(* PLC project PLC_Programming_With_ST.project, TK TC6_v0200_Example3 v3.0 *)
(* stored: creationDateTime 2019-09-29T20:50:27.2524554, modificationDateTime 2020-05-23T11:25:38.4825215 *)

TYPE OnOff_ConstructorLIO : STRUCT
  Opened : BOOL;  (* Object is opened *)
  Closed : BOOL;  (* Object is closed *)
  PositionError : BOOL;  (* TRUE: Object has position error *)
END_STRUCT;
END_TYPE

TYPE dint8 : STRUCT
  first : DINT;
  second : DINT;
  third : DINT;
  fourth : DINT;
  fifth : DINT;
  sixth : DINT;
  seventh : DINT;
  eight : DINT;
END_STRUCT;
END_TYPE

TYPE MotorPump : STRUCT
  Running : BOOL;
  Fail : BOOL;
  DiffPress : BOOL;
END_STRUCT;
END_TYPE

TYPE MotorVentilator : STRUCT
  qMotor : BOOL;
  iOverheatProtection : BOOL;
  iOvercurrentProtection : BOOL;
  iMotorFailOther : BOOL;
  qLamp_Local : BOOL;
  iEmcy_Stop : BOOL := TRUE;
  iStart_Local : BOOL;
  iStop_Local : BOOL;
END_STRUCT;
END_TYPE

TYPE PrometnoSvjetlo : STRUCT
  ZelenoSvjetlo : BOOL;
  ZutoSvjetlo : BOOL;
  CrvenoSvjetlo : BOOL;
  PjesakovoDugme : BOOL;
END_STRUCT;
END_TYPE

{attribute 'qualified_only'}
VAR_GLOBAL  (* MixingTankGVL *)
  PushButtonStart : BOOL;  (* DIGITAL INPUT Naredba operator za start sustava *)
  PushButtonStop : BOOL;  (* DIGITAL INPUT Naredba operator za stop sustava *)
  Pump1StartCmd : BOOL;  (* DIGITAL OUTPUT Naredba automatike za start pumpe 1 *)
  Pump1StopCmd : BOOL;  (* DIGITAL OUTPUT Naredba automatike za stop pumpe 1 *)
  Pump1Running : BOOL;  (* DIGITAL INPUT Indikacija pokrenutog status pumpe 1 *)
  Pump2StartCmd : BOOL;  (* DIGITAL OUTPUT Naredba automatike za start pumpe 2 *)
  Pump2StopCmd : BOOL;  (* DIGITAL OUTPUT Naredba automatike za stop pumpe 2 *)
  Pump2Running : BOOL;  (* DIGITAL INPUT Indikacija pokrenutog status pumpe 2 *)
  DrainValveOpenCmd : BOOL;  (* DIGITAL OUTPUT Naredba automatike za otvaranje ventila za odvod *)
  DrainValveCloseCmd : BOOL;  (* DIGITAL OUTPUT Naredba automatike za zatvaranje ventila za odvod *)
  DrainValveClosed : BOOL;  (* DIGITAL INPUT Indikacija zatvorenog stanja odvodnog ventila *)
  DrainValveOpened : BOOL;  (* DIGITAL INPUT Indikacija otvorenog stanja odvodnog ventila *)
  TankLevel : REAL;  (* REAL VALUE Trenutna razina tanka u postocima *)
END_VAR

{attribute 'qualified_only'}
VAR_GLOBAL  (* Task02GVL *)
  HorizontalS1 : BOOL;  (* Configuration Inputs *)
  HorizontalS2 : BOOL;
  VerticalS1 : BOOL;
  VerticalS2 : BOOL;
  ManUp : BOOL;
  ManDown : BOOL;
  ManRight : BOOL;
  ManLeft : BOOL;
  ManUpRight : BOOL;
  ManUpLeft : BOOL;
  ManDownRight : BOOL;
  ManDownLeft : BOOL;
  Reset : BOOL;
  HorizontalRight : BOOL;  (* Outputs *)
  HorizontalLeft : BOOL;
  VerticalUp : BOOL;
  VerticalDown : BOOL;
END_VAR

{attribute 'qualified_only'}
VAR_GLOBAL  (* Task03GVL *)
  cfgPeriodTime : TIME := TIME#1m24s0ms;  (* Configuration *)
  cfgStartDirection : DINT := 0;
  TLight1Red : BOOL;  (* DIGITAL OUTPUT Activate red light traffic light 1 *)
  TLight1Yellow : BOOL;  (* DIGITAL OUTPUT Activate yellow light traffic light 1 *)
  TLight1Green : BOOL;  (* DIGITAL OUTPUT Activate green light traffic light 1 *)
  TLight2Red : BOOL;  (* DIGITAL OUTPUT Activate red light traffic light 2 *)
  TLight2Yellow : BOOL;  (* DIGITAL OUTPUT Activate yellow light traffic light 2 *)
  TLight2Green : BOOL;  (* DIGITAL OUTPUT Activate green light traffic light 2 *)
  TLight3Red : BOOL;  (* DIGITAL OUTPUT Activate red light traffic light 3 *)
  TLight3Yellow : BOOL;  (* DIGITAL OUTPUT Activate yellow light traffic light 3 *)
  TLight3Green : BOOL;  (* DIGITAL OUTPUT Activate green light traffic light 3 *)
  TLight4Red : BOOL;  (* DIGITAL OUTPUT Activate red light traffic light 4 *)
  TLight4Yellow : BOOL;  (* DIGITAL OUTPUT Activate yellow light traffic light 4 *)
  TLight4Green : BOOL;  (* DIGITAL OUTPUT Activate green light traffic light 4 *)
END_VAR



{attribute 'qualified_only'}
VAR_GLOBAL  (* Task06GVL *)
  JoyUp : BOOL;  (* Configuration Inputs *)
  JoyDown : BOOL;
  JoyRight : BOOL;
  JoyLeft : BOOL;
  JoyUpRight : BOOL;
  JoyUpLeft : BOOL;
  JoyDownRight : BOOL;
  JoyDownLeft : BOOL;
  EmcyStop : BOOL;
  RightLimit : BOOL;
  LeftLimit : BOOL;
  UpperLimit : BOOL;
  LowerLimit : BOOL;
  MotorLeft : BOOL;  (* Outputs *)
  MotorRight : BOOL;
  CraneDown : BOOL;
  CraneUp : BOOL;
END_VAR





PROGRAM FOR_Loop
  VAR CONSTANT
    ARR_SIZE : USINT := 9;  (* Size of the cube *)
  END_VAR
  VAR
    vType : USINT := 0;
    data : ARRAY[0..ARR_SIZE, 0..ARR_SIZE] OF BOOL;  (* Data for iteration *)
    i : USINT;  (* Iterators *)
    j : USINT;  (* Iterators *)
    vIncStep : BOOL;  (* Support functionalities *)
    vDecStep : BOOL;
    vStepTime : TIME := TIME#1s0ms;
    vStepTimeChange : TIME := TIME#100ms;
    Stepper : BLINK;
  END_VAR

            CASE vType OF
	0: (*FOR LOOP*)
		(*Loop over everything, set always to inverse*)
		FOR i:=0 TO ARR_SIZE DO
			(*Go through all the columns of this row*)
			FOR j:=0 TO ARR_SIZE DO
				data[i,j] := NOT data[i,j];
			END_FOR
		END_FOR
		
	1: (*WHILE LOOP*)
		(*Loop over everything, set always to inverse*)
		WHILE i <= ARR_SIZE DO
			(*Go trough all the columns*)
			WHILE j <= ARR_SIZE DO
				data[i,j] := NOT data[i,j];
				j := j + 1;
			END_WHILE
			j := 0;
			(*After each column, increase row by 1*)
			i := i + 1;			
		END_WHILE
		(*If we ended up here, that means we went throguh all the elements,
		so we can reset and start all over*)
		i := 0;
		j := 0;
	
	2: (*Repeat loop*)
		(*Repeat loop executes atleast once*)
		REPEAT

			REPEAT
				data[i,j] := NOT data[i,j];
				j := j + 1;
			UNTIL
				j > ARR_SIZE
			END_REPEAT
			j := 0;
			i := i + 1;
		UNTIL
			i > ARR_SIZE
		END_REPEAT
		i := 0;
		j := 0;
		
	3: (*Cycle loop on 100 ms*)
		data[i,j] := NOT data[i,j];
		j := j + 1;
		IF j > ARR_SIZE THEN
			j:=0;
			i := i + 1;
			IF i > ARR_SIZE THEN
				i := 0;
			END_IF
		END_IF
		
	4: (*Pulse/Trigger loop*)
		IF Stepper.OUT THEN
			data[i,j] := NOT data[i,j];
			j := j + 1;
			IF j > ARR_SIZE THEN
				j:=0;
				i := i + 1;
				IF i > ARR_SIZE THEN
					i := 0;
				END_IF
			END_IF
		END_IF
	
	5: (*Reset - Set all to false*)
		MEMUtils.MemSet(ADR(data),0, SIZEOF(data));
END_CASE

(*Support functionality*)
(*Step speed*)
IF vIncStep THEN
	vStepTime := LIMIT(T#0.1S, vStepTime + vStepTimeChange, T#10S);
ELSIF vDecStep THEN
	vStepTime := LIMIT(T#0.1S, vStepTime - vStepTimeChange, T#10S);
END_IF
Stepper(ENABLE:= TRUE, TIMELOW:= vStepTime, TIMEHIGH:= T#100MS);
          
END_PROGRAM

FUNCTION_BLOCK CollisionDetection
  VAR_INPUT
    xcor1 : REAL := 0;  (* X Coordinate of object 1 *)
    ycor1 : REAL := 0;  (* Y Coordinate of object 1 *)
    height1 : REAL := 0;  (* Height of object 1 *)
    width1 : REAL := 0;  (* Width of object 1 *)
    xcor2 : REAL := 0;  (* X Coordinate of object 2 *)
    ycor2 : REAL := 0;  (* Y Coordinate of object 2 *)
    height2 : REAL := 0;  (* Height of object 1 *)
    width2 : REAL := 0;  (* Width of object 1 *)
  END_VAR
  VAR_OUTPUT
    isCollision : BOOL := FALSE;
  END_VAR

            IF xcor1 < (xcor2 + width2) AND
   (xcor1 + width1) > xcor2 AND
   ycor1 < (ycor2 + height2) AND
  ( height1 + ycor1) > ycor2 THEN
   isCollision := TRUE;
ELSE
	isCollision := FALSE;
END_IF
          
END_FUNCTION_BLOCK

FUNCTION CONCAT2 : STRING
  VAR_INPUT
    STR : ARRAY[0..19] OF STRING;  (* String array filled with characters to concatenate *)
  END_VAR
  VAR
    vStr : STRING := '';
    i : UINT := 0;
    vSize : UINT;
  END_VAR

            vStr := '';
vSize :=(SIZEOF(STR)/81);

FOR i:=0 TO vSize - 1 BY 1 DO
	IF STR[i] <> '' THEN
		vStr := CONCAT(vStr, STR[i]);
	END_IF
END_FOR
CONCAT2 := vStr;
          
END_FUNCTION

PROGRAM PLC_PRG_1
  VAR
    Start_Switch : BOOL;
    Bottle : BOOL;
    UpperLimitSwitch : BOOL := TRUE;
    ConveyorBeltPut : BOOL;
    ConveyorBeltSimPut : TON;
    TimeSimConvey : TIME := TIME#2s0ms;
    MotorDown : BOOL;
    LowerLimitSwitch : BOOL;
    MotorUp : BOOL;
    MovingDownSim : TON;
    TimeDownSim : TIME := TIME#4s0ms;
    ElapsedTimeDown : TIME;
    TimeCheck : TIME := TIME#0ms;
    BottleStamped : BOOL;
    MovingUpSim : TON;
    TimeUpSim : TIME := TIME#4s0ms;
    ElapsedTimeUp : TIME;
    ConveyorBeltRemove : BOOL;
    ConveyorBeltRemoveSim : TON;
    ConveyorBeltMotor : BOOL;
  END_VAR

            IF Start_Switch THEN

	(* Putting new bottle under the marker if there isnt any *)
	IF NOT Bottle AND UpperLimitSwitch THEN
		ConveyorBeltPut := TRUE;
	ELSE
		ConveyorBeltPut := FALSE;
	END_IF;

	(*Simulating the conveyor belt putting new bottle in*)
	ConveyorBeltSimPut(IN:= ConveyorBeltPut, PT:= TimeSimConvey);

	IF ConveyorBeltSimPut.Q THEN
		Bottle := TRUE;
	END_IF;

	MotorDown := Bottle AND NOT LowerLimitSwitch AND NOT MotorUp;
	(*Simulating the movement of the motor down and engaging the limit switches*)
	MovingDownSim(IN := MotorDown, PT := TimeDownSim, ET => ElapsedTimeDown);

	IF MovingDownSim.ET <> TimeCheck THEN
		UpperLimitSwitch := FALSE;
	END_IF;

	IF MovingDownSim.Q THEN
		LowerLimitSwitch := TRUE;
		BottleStamped :=TRUE;
	END_IF;

	MotorUp := BottleStamped AND NOT UpperLimitSwitch AND NOT MotorDown;
	(*Simulating the movement of the motor up and engaging the limit switches*)
	MovingUpSim(IN := MotorUp,PT := TimeUpSim, ET=>ElapsedTimeUp);

	IF MovingUpSim.ET <> TimeCheck THEN
		LowerLimitSwitch := FALSE;
	END_IF;

	IF MovingUpSim.Q THEN
		UpperLimitSwitch := TRUE;
	END_IF;

	IF BottleStamped AND UpperLimitSwitch THEN
		ConveyorBeltRemove := TRUE;
		(*Simulating the rotation of the conveyor and removing the bottles that is stamped*)
		ConveyorBeltRemoveSim(IN := ConveyorBeltRemove, PT := TimeSimConvey );
		IF ConveyorBeltRemoveSim.Q THEN
			Bottle := FALSE;
			BottleStamped := FALSE;
		END_IF;
	ELSE
		ConveyorBeltRemove := FALSE;
	END_IF;

	ConveyorBeltMotor := ConveyorBeltRemove OR ConveyorBeltPut;

END_IF;
(*
IF Start_Switch THEN

	IF  UpperLimitSwitch
		AND NOT LowerLimitSwitch
		AND NOT CylinderUpMotor
		THEN
			CylinderDownMotor := TRUE;
	END_IF;

	UpperLSWDelay(IN:=CylinderDownMotor, PT:=T#10S);
	IF 	UpperLSWDelay.Q
	THEN
		LowerLimitSwitch := TRUE;
	END_IF;

	IF  LowerLimitSwitch
	THEN
		CylinderDownMotor:= FALSE;
	END_IF;

	IF 	UpperLimitSwitch
	THEN
		CylinderUpMotor := FALSE;
	END_IF;

	IF 			 LowerLimitSwitch
		AND NOT  UpperLimitSwitch
	THEN
				 CylinderUpMotor := TRUE;
	END_IF;
	
	LowerLSWDelay(IN:=CylinderUpMotor, PT:=T#10S);
	IF 	LowerLSWDelay.Q
	THEN
		UpperLimitSwitch := TRUE;
	END_IF;

	IF UpperLimitSwitch
	THEN
		LowerLimitSwitch := FALSE;
	ELSE IF LowerLimitSwitch
	THEN
 	UpperLimitSwitch:FALSE;
	END_IF;

END_IF;
*)

          
END_PROGRAM

FUNCTION_BLOCK Motor_Model
  VAR_INPUT
    CBActivated : BOOL := FALSE;
    LineVoltage : REAL := 440;
    cfgNominalPower : REAL := 12;  (* kW *)
    cfgPowerFactor : REAL := 0.83;
    Frequency : REAL := 60;
    cfgNoOfPoles : DINT := 4;
    cfgSpeedUpRate : REAL := 800;
    cfgSpeedDownRate : REAL := 800;
    simShortCircuit : BOOL := FALSE;
  END_VAR
  VAR_OUTPUT
    CurrentL1 : LREAL := 0;
    CurrentL2 : LREAL := 0;
    CurrentL3 : LREAL := 0;
    Speed : REAL := 0;
    Status : ARRAY[0..10] OF BOOL;
  END_VAR
  VAR
    vNs : REAL;
    vPhaseCurrent : REAL := 0;
    SpeedRamp : RAMP_REAL;
    SpeedBlink : BLINK;
    vBlinkTime : REAL;
    vBlinker : BOOL;
    vApparentPower_kVA : REAL;
  END_VAR

            Status[0] := CBActivated;;

vApparentPower_kVA := cfgNominalPower/(3*cfgPowerFactor);

vPhaseCurrent := (vApparentPower_kVA*1000)/LineVoltage;

CurrentL1 := (vPhaseCurrent/SQRT(3)+(BOOL_TO_REAL(simShortCircuit)*250))*BOOL_TO_REAL(Status[0]);
CurrentL2 := (vPhaseCurrent/SQRT(3)+(BOOL_TO_REAL(simShortCircuit)*250))*BOOL_TO_REAL(Status[0]);
CurrentL3 := (vPhaseCurrent/SQRT(3)+(BOOL_TO_REAL(simShortCircuit)*250))*BOOL_TO_REAL(Status[0]);

vNs := ((120 *Frequency)/DINT_TO_REAL(cfgNoOfPoles))*BOOL_TO_REAL(Status[0]);

SpeedRamp(
	IN:= vNs, 
	ASCEND:= cfgSpeedUpRate, 
	DESCEND:= cfgSpeedDownRate, 
	TIMEBASE:= T#2S, 
	OUT=>Speed);
	
vBlinkTime := 100000/MAX(1,Speed);

SpeedBlink(ENABLE:= vBlinkTime < 100000, TIMELOW:= REAL_TO_TIME(vBlinkTime), TIMEHIGH:= REAL_TO_TIME(vBlinkTime), OUT=> Status[1]);
          
END_FUNCTION_BLOCK

FUNCTION_BLOCK On_Off_Constructor
  VAR_INPUT
    iOpenedFB : BOOL;  (* IO Open signal feedback from the valve *)
    iClosedFB : BOOL;  (* IO Close signal feedback from the valve *)
    cfgPositionErrorDelay : TIME := TIME#10s0ms;  (* Position error alarm delay *)
    cfgFBs : DWORD := 3;  (* B0 - Opened signal in use, B1 - Closed signal in use *)
  END_VAR
  VAR_OUTPUT
    LIO : OnOff_ConstructorLIO;  (* Communication structure to higher logic *)
    HMI : OnOff_ConstructorLIO;  (* Communication structure to HMI *)
  END_VAR
  VAR
    PositionErrorDelay : TON;  (* Position error alarm delay *)
    vPositionErrorOld : BOOL;  (* Event memory: Position error *)
    vOpenedOld : BOOL;  (* Event memory: Opened *)
    vClosedOld : BOOL;  (* Event memory: Closed *)
  END_VAR

            (* Handle IOs depending on CFG *)
IF cfgFBs.0 AND cfgFBs.1 THEN
	LIO.Closed := iClosedFB;
	LIO.Opened := iOpenedFB;
ELSIF cfgFBs.0 THEN
	LIO.Closed := NOT iOpenedFB;
	LIO.Opened := iOpenedFB;
ELSIF cfgFBs.1 THEN
	LIO.Closed := iClosedFB;
	LIO.Opened := NOT iClosedFB;
ELSE
	(* Invalid configuration *)
END_IF;

(* Alarm management *)
(* Position error *)
PositionErrorDelay(
	IN:= LIO.Closed AND LIO.Opened OR NOT (LIO.Closed OR LIO.Opened),
	PT:= cfgPositionErrorDelay,
	Q  => LIO.PositionError);

(* Event management *)
(* Breaker opened *)
IF LIO.Opened AND NOT vOpenedOld THEN
	(* Call event *)
END_IF

(* Breaker closed *)
IF LIO.Closed AND NOT vClosedOld THEN
	(* Call event *)
END_IF
(* Position error *)
IF LIO.PositionError AND NOT vPositionErrorOld THEN
	(* Call event *)
END_IF

(* Communicate status to HMI *)	
HMI := LIO;


 
          
END_FUNCTION_BLOCK

FUNCTION_BLOCK OnOffValve_Model
  VAR_INPUT
    OpenCmd : BOOL;  (* Command to open the valve *)
    CloseCmd : BOOL;  (* Command to close the valve *)
    cfgOpeningTime : TIME := TIME#5s0ms;  (* Time it take to open the valve *)
    cfgClosingTime : TIME := TIME#5s0ms;  (* Time it take to close the valve *)
    simOpenFail : BOOL;  (* Simulated open fail when true *)
    simCloseFail : BOOL;  (* Simulated close fail when true *)
  END_VAR
  VAR_OUTPUT
    Opened : BOOL;
    Closed : BOOL;
  END_VAR
  VAR
    OpenTime : TON;
    CloseTime : TON;
  END_VAR

            (* Description of action:
If the open/close signal comes the valve opens/closes in designated time *)

OpenTime(IN:= OpenCmd AND NOT Opened, PT:=cfgOpeningTime);
CloseTime(IN:= CloseCmd AND NOT Closed, PT:=cfgClosingTime);

IF Opened AND CloseCmd THEN
	Opened := FALSE;
ELSIF OpenTime.Q AND NOT simOpenFail THEN
	Opened := TRUE;
END_IF

IF Closed AND OpenCmd THEN
	Closed := FALSE;
ELSIF CloseTime.Q AND NOT simCloseFail THEN
	Closed := TRUE;
END_IF
          
END_FUNCTION_BLOCK

FUNCTION_BLOCK OnOffValve_Object
  VAR_INPUT
    iOpenedFB : BOOL;  (* IO Open signal feedback from the valve *)
    iClosedFB : BOOL;  (* IO Close signal feedback from the valve *)
    OpenAutoCmd : BOOL;  (* Open cmd from program logic *)
    CloseAutoCmd : BOOL;  (* Close cmd from program logic *)
    OpenCmdHMI : BOOL;  (* Open cmd from HMI *)
    CloseCmdHMI : BOOL;  (* Close cmd from HMI *)
    SetToAuto : BOOL;  (* Sets valve control to auto mode *)
    SetToMan : BOOL;  (* Sets valve control to manual mode *)
    cfgOpenFailDelay : TIME := TIME#6s0ms;  (* Open fail delay *)
    cfgCloseFailDelay : TIME := TIME#6s0ms;  (* Close fail delay *)
    cfgPositionErrorDelay : TIME := TIME#10s0ms;  (* Position error delay *)
    cfgFBs : DWORD := 16#3;  (* B0 - Opened signal in use, B1 - Closed signal in use *)
  END_VAR
  VAR_OUTPUT
    ValveStatus : ARRAY[1..20] OF DINT;  (* 1:Open/Closed/InTransit, 2:OpenFail, 3:CloseFail, 4:FBError, 5:Control Position, 6:OpenCmd, 7:CloseCmd *)
    ValveIcon : STRING;
    qOpenCmd : BOOL;  (* IO Open command signal *)
    qCloseCmd : BOOL;  (* IO Close command signal *)
  END_VAR
  VAR
    ObjConstructor : On_Off_Constructor;  (* Base building block of this object *)
    OpenFail : TON;
    CloseFail : TON;
    vControlPosition : DINT;
    vOpenCmd : BOOL;
    vCloseCmd : BOOL;
  END_VAR

            (* Handle base constructor *)
ObjConstructor(
	iOpenedFB := iOpenedFB,
	iClosedFB := iClosedFB,
	cfgPositionErrorDelay := cfgPositionErrorDelay,
	cfgFBs := cfgFBs);

(* Control position *)
(* Auto/Man setting should be rtrig or non holding button *)
IF SetToAuto AND NOT SetToMan THEN
	vControlPosition := 1;
ELSIF SetToMan THEN
	vControlPosition := 0;
END_IF

IF NOT(OpenFail.Q OR CloseFail.Q) THEN
	IF vControlPosition = 1 THEN
		vOpenCmd := (vOpenCmd OR OpenAutoCmd) AND NOT ObjConstructor.LIO.Opened;
		vCloseCmd := (vCloseCmd OR CloseAutoCmd) AND NOT ObjConstructor.LIO.Closed;
	ELSIF vControlPosition = 0 THEN
		vOpenCmd := (vOpenCmd OR OpenCmdHMI) AND NOT ObjConstructor.LIO.Opened;
		vCloseCmd := (vCloseCmd OR CloseCmdHMI) AND NOT ObjConstructor.LIO.Closed;
	ELSE
		vOpenCmd := FALSE;
		vCloseCmd := FALSE;	
	END_IF
ELSE
		vOpenCmd := FALSE;
		vCloseCmd := FALSE;		
END_IF

OpenFail(IN:= vOpenCmd AND NOT ObjConstructor.LIO.Opened, PT:= cfgOpenFailDelay);
CloseFail(IN:= vCloseCmd AND NOT ObjConstructor.LIO.Closed, PT:= cfgCloseFailDelay);

qOpenCmd := vOpenCmd AND NOT (OpenFail.Q OR ObjConstructor.LIO.Opened OR ObjConstructor.LIO.PositionError);
qCloseCmd := vCloseCmd AND NOT (CloseFail.Q OR ObjConstructor.LIO.Closed OR ObjConstructor.LIO.PositionError);

ValveStatus[1] := BOOL_TO_DINT(ObjConstructor.LIO.Opened) + 2*BOOL_TO_DINT(ObjConstructor.LIO.Closed);
ValveStatus[2] := BOOL_TO_DINT(OpenFail.Q);
ValveStatus[3] := BOOL_TO_DINT(CloseFail.Q);
ValveStatus[4] := BOOL_TO_DINT(ObjConstructor.LIO.PositionError);
ValveStatus[5] := vControlPosition;
ValveStatus[6] := BOOL_TO_DINT(qOpenCmd);
ValveStatus[7] := BOOL_TO_DINT(qCloseCmd);

IF ValveStatus[1] = 1 THEN
	ValveIcon := 'Valve1';
ELSIF ValveStatus[1] = 2 THEN
	ValveIcon := 'Valve2';
ELSE
	ValveIcon := 'Valve3';
END_IF


          
END_FUNCTION_BLOCK

PROGRAM PriorityPOU
  VAR
    SortPriority : PrioritySort;
    SwapSequence1 : Swapper;
    SwapSequence2 : Swapper;
    FPSequenceChangeTimer : TON;
    vEngineSequence : dint8;
    vFPSequence : dint8;
    vPPSequence : dint8;
    vModeManagerSequence : dint8;
    vApplyNewSequence : BOOL;
    vApplyButtonPermission : BOOL;
    vNewSequence : dint8;
    vSequenceIsSame : BOOL;
    vValidStartSequenceSum : LREAL;
    vEngineSequenceSum : LREAL;
    vFPSequenceSum : LREAL;
    vFPSequenceInvalid : BOOL;
    vApplyButton2Permission : BOOL;
  END_VAR
  VAR RETAIN
    vRestarted : BOOL := FALSE;
    vInvalidSequence : BOOL;
  END_VAR

            
IF NOT vRestarted OR vInvalidSequence THEN
	(* Reinitialize priority list *)
	vEngineSequence.first := 1;
	vEngineSequence.second := 2;
	vEngineSequence.third  := 3;
	vEngineSequence.fourth := 4;
	vEngineSequence.fifth := 5;
	vEngineSequence.sixth := 6;
	vEngineSequence.seventh := 7;
	vEngineSequence.eight := 8;
	vFPSequence := vEngineSequence;
	vRestarted := TRUE;
END_IF

(* Determine correct sequence sum *)
vValidStartSequenceSum := EXPT(2,1)
						+ EXPT(2,2)
						+ EXPT(2,3)
                        + EXPT(2,4)
						+ EXPT(2,5)
						+ EXPT(2,6)
						+ EXPT(2,7)
						+ EXPT(2,8);

(* Constantly check engine sequence to make sure it is correct *)
vEngineSequenceSum := EXPT(2,vEngineSequence.first)
					+ EXPT(2,vEngineSequence.second)
					+ EXPT(2,vEngineSequence.third)
                    + EXPT(2,vEngineSequence.fourth)
				    + EXPT(2,vEngineSequence.fifth)
				    + EXPT(2,vEngineSequence.sixth)
					+ EXPT(2,vEngineSequence.seventh)
					+ EXPT(2,vEngineSequence.eight);
					
vInvalidSequence := vEngineSequenceSum <> vValidStartSequenceSum;

(* Faceplate start sequence handling *)
vSequenceIsSame :=  vEngineSequence.first = vFPSequence.first
				AND vEngineSequence.second = vFPSequence.second
				AND vEngineSequence.third = vFPSequence.third
				AND vEngineSequence.fourth = vFPSequence.fourth
				AND vEngineSequence.fifth = vFPSequence.fifth
				AND vEngineSequence.sixth = vFPSequence.sixth
				AND vEngineSequence.seventh = vFPSequence.seventh
				AND vEngineSequence.eight = vFPSequence.eight;

vFPSequenceSum := EXPT(2,vFPSequence.first)
				+ EXPT(2,vFPSequence.second)
				+ EXPT(2,vFPSequence.third)
                + EXPT(2,vFPSequence.fourth)
				+ EXPT(2,vFPSequence.fifth)
				+ EXPT(2,vFPSequence.sixth)
				+ EXPT(2,vFPSequence.seventh)
				+ EXPT(2,vFPSequence.eight);
				
vFPSequenceInvalid := vFPSequenceSum <> vValidStartSequenceSum;	
			
FPSequenceChangeTimer(IN:= NOT vSequenceIsSame OR vFPSequenceInvalid, PT:=T#15S);
IF FPSequenceChangeTimer.Q THEN
	vFPSequence := vEngineSequence;
END_IF;	
		
(* Swapper function 
- swaps places with the selected number*)
SwapSequence1(Enable:= NOT vSequenceIsSame, SequenceIN:= vFPSequence, SequenceOut => vFPSequence);

(* Functionality:
- Takes care of reseting invalid seq
- Applies requests
- converts to engine format
*)
SortPriority(
	EngineSequenceIN := vEngineSequence,
	RequestSequence1:= vFPSequence,
	RequestSequence1Permission:= NOT vFPSequenceInvalid,
	RequestSequence1Apply:= vApplyNewSequence,
	RequestSequence2:= vPPSequence,
	RequestSequence2Permission:= FALSE,
	RequestSequence2Apply:= FALSE,
	RequestSequence1ApplyPermission=> vApplyButtonPermission,
	RequestSequence2ApplyPermission=> vApplyButton2Permission,
	RequestSequence1OUT=> vFPSequence,
	RequestSequence2OUT=> vPPSequence,
	EngineSequenceOUT=> vEngineSequence);

          
END_PROGRAM

FUNCTION_BLOCK PrioritySort
  VAR_INPUT
    EngineSequenceIN : dint8;
    RequestSequence1 : dint8;
    RequestSequence1Permission : BOOL;
    RequestSequence1Apply : BOOL;
    RequestSequence2 : dint8;
    RequestSequence2Permission : BOOL;
    RequestSequence2Apply : BOOL;
  END_VAR
  VAR_OUTPUT
    RequestSequence1ApplyPermission : BOOL;
    RequestSequence2ApplyPermission : BOOL;
    RequestSequence1OUT : dint8;
    RequestSequence2OUT : dint8;
    EngineSequenceOUT : dint8;
  END_VAR
  VAR
    v1stSeqDifferent : BOOL;
    v2ndSeqDifferent : BOOL;
  END_VAR

            (* Compare sequences *)
v1stSeqDifferent := RequestSequence1.first <> EngineSequenceIN.first
				OR  RequestSequence1.second <> EngineSequenceIN.second
				OR  RequestSequence1.third <> EngineSequenceIN.third
				OR  RequestSequence1.fourth <> EngineSequenceIN.fourth
				OR  RequestSequence1.fifth <> EngineSequenceIN.fifth
				OR  RequestSequence1.sixth <> EngineSequenceIN.sixth
				OR  RequestSequence1.seventh <> EngineSequenceIN.seventh
				OR  RequestSequence1.eight <> EngineSequenceIN.eight;

v2ndSeqDifferent := RequestSequence2.first <> EngineSequenceIN.first
				OR  RequestSequence2.second <> EngineSequenceIN.second
				OR  RequestSequence2.third <> EngineSequenceIN.third
				OR  RequestSequence2.fourth <> EngineSequenceIN.fourth
				OR  RequestSequence2.fifth <> EngineSequenceIN.fifth
				OR  RequestSequence2.sixth <> EngineSequenceIN.sixth
				OR  RequestSequence2.seventh <> EngineSequenceIN.seventh
				OR  RequestSequence2.eight <> EngineSequenceIN.eight;

IF v1stSeqDifferent AND RequestSequence1Permission AND RequestSequence1Apply THEN
	EngineSequenceOUT := RequestSequence1;
	RequestSequence2OUT := RequestSequence1;
	
ELSIF v2ndSeqDifferent AND RequestSequence2Permission AND RequestSequence2Apply THEN
	EngineSequenceOUT := RequestSequence2;
	RequestSequence1OUT := RequestSequence2;
	
ELSE
	(* Basically do nothing, copy parameters *)
	EngineSequenceOUT := EngineSequenceIN;
	RequestSequence1OUT := RequestSequence1;
	RequestSequence2OUT := RequestSequence2;
END_IF

(* Send out permissions *)
RequestSequence1ApplyPermission:= RequestSequence1Permission AND NOT RequestSequence2Apply;
RequestSequence2ApplyPermission:= RequestSequence2Permission AND NOT RequestSequence1Apply;
          
END_FUNCTION_BLOCK

FUNCTION_BLOCK Swapper
  VAR_INPUT
    Enable : BOOL;
    SequenceIn : dint8;
  END_VAR
  VAR_OUTPUT
    SequenceOut : dint8;
  END_VAR
  VAR
    vTemp : DINT;
  END_VAR

            IF Enable THEN
	(* Check if any of the positions have changed values *)
	IF SequenceIN.first <> SequenceOut.first THEN
		(* If this position changed, save the old position and apply new one to its place *)
		vTemp:= SequenceOut.first;
		SequenceOut.first := SequenceIN.first;
		(* Find the position where the same number is and write temp there
		but skip this position *)
		IF SequenceIN.first = SequenceOut.second THEN
			SequenceOut.second := vTemp;
		ELSIF SequenceIN.first = SequenceOut.third THEN
			SequenceOut.third := vTemp;
		ELSIF SequenceIN.first = SequenceOut.fourth THEN
			SequenceOut.fourth := vTemp;
		ELSIF SequenceIN.first = SequenceOut.fifth THEN
			SequenceOut.fifth := vTemp;
		ELSIF SequenceIN.first = SequenceOut.sixth THEN
			SequenceOut.sixth := vTemp;
		ELSIF SequenceIN.first = SequenceOut.seventh THEN
			SequenceOut.seventh := vTemp;
		ELSIF SequenceIN.first = SequenceOut.eight THEN
			SequenceOut.eight := vTemp;
		END_IF
	ELSIF SequenceIN.second <> SequenceOut.second THEN
		vTemp:= SequenceOut.second;
		SequenceOut.second := SequenceIN.second;
		(* Find the index where the same number is and write temp there
		but skip this position *)
		IF SequenceIN.second = SequenceOut.first THEN
			SequenceOut.first := vTemp;
		ELSIF SequenceIN.second = SequenceOut.third THEN
			SequenceOut.third := vTemp;
		ELSIF SequenceIN.second = SequenceOut.fourth THEN
			SequenceOut.fourth := vTemp;
		ELSIF SequenceIN.second = SequenceOut.fifth THEN
			SequenceOut.fifth := vTemp;
		ELSIF SequenceIN.second = SequenceOut.sixth THEN
			SequenceOut.sixth := vTemp;
		ELSIF SequenceIN.second = SequenceOut.seventh THEN
			SequenceOut.seventh := vTemp;
		ELSIF SequenceIN.second = SequenceOut.eight THEN
			SequenceOut.eight := vTemp;
		END_IF
	ELSIF SequenceIN.third <> SequenceOut.third THEN
			vTemp:= SequenceOut.third;
		SequenceOut.third := SequenceIN.third;
		(* Find the index where the same number is and write temp there
		but skip this position *)
		IF SequenceIN.third = SequenceOut.first THEN
			SequenceOut.first := vTemp;
		ELSIF SequenceIN.third = SequenceOut.second THEN
			SequenceOut.second := vTemp;
		ELSIF SequenceIN.third = SequenceOut.fourth THEN
			SequenceOut.fourth := vTemp;
		ELSIF SequenceIN.third = SequenceOut.fifth THEN
			SequenceOut.fifth := vTemp;
		ELSIF SequenceIN.third = SequenceOut.sixth THEN
			SequenceOut.sixth := vTemp;
		ELSIF SequenceIN.third = SequenceOut.seventh THEN
			SequenceOut.seventh := vTemp;
		ELSIF SequenceIN.third = SequenceOut.eight THEN
			SequenceOut.eight := vTemp;
		END_IF
	ELSIF SequenceIN.fourth <> SequenceOut.fourth THEN
			vTemp:= SequenceOut.fourth;
		SequenceOut.fourth := SequenceIN.fourth;
		(* Find the index where the same number is and write temp there
		but skip this position *)
		IF SequenceIN.third = SequenceOut.first THEN
			SequenceOut.first := vTemp;
		ELSIF SequenceIN.fourth = SequenceOut.second THEN
			SequenceOut.second := vTemp;
		ELSIF SequenceIN.fourth = SequenceOut.third THEN
			SequenceOut.third := vTemp;
		ELSIF SequenceIN.fourth = SequenceOut.fifth THEN
			SequenceOut.fifth := vTemp;
		ELSIF SequenceIN.fourth = SequenceOut.sixth THEN
			SequenceOut.sixth := vTemp;
		ELSIF SequenceIN.fourth = SequenceOut.seventh THEN
			SequenceOut.seventh := vTemp;
		ELSIF SequenceIN.fourth = SequenceOut.eight THEN
			SequenceOut.eight := vTemp;
		END_IF
	ELSIF SequenceIN.fifth <> SequenceOut.fifth THEN
			vTemp:= SequenceOut.fifth;
		SequenceOut.fifth := SequenceIN.fifth;
		(* Find the index where the same number is and write temp there
		but skip this position *)
		IF SequenceIN.fifth = SequenceOut.first THEN
			SequenceOut.first := vTemp;
		ELSIF SequenceIN.fifth = SequenceOut.second THEN
			SequenceOut.second := vTemp;
		ELSIF SequenceIN.fifth = SequenceOut.third THEN
			SequenceOut.third := vTemp;
		ELSIF SequenceIN.fifth = SequenceOut.fourth THEN
			SequenceOut.fourth := vTemp;
		ELSIF SequenceIN.fifth = SequenceOut.sixth THEN
			SequenceOut.sixth := vTemp;
		ELSIF SequenceIN.fifth = SequenceOut.seventh THEN
			SequenceOut.seventh := vTemp;
		ELSIF SequenceIN.fifth = SequenceOut.eight THEN
			SequenceOut.eight := vTemp;
		END_IF
	ELSIF SequenceIN.sixth <> SequenceOut.sixth THEN
			vTemp:= SequenceOut.sixth;
		SequenceOut.sixth := SequenceIN.sixth;
		(* Find the index where the same number is and write temp there
		but skip this position *)
		IF SequenceIN.sixth = SequenceOut.first THEN
			SequenceOut.first := vTemp;
		ELSIF SequenceIN.sixth = SequenceOut.second THEN
			SequenceOut.second := vTemp;
		ELSIF SequenceIN.sixth = SequenceOut.third THEN
			SequenceOut.third := vTemp;
		ELSIF SequenceIN.sixth = SequenceOut.fourth THEN
			SequenceOut.fourth := vTemp;
		ELSIF SequenceIN.sixth = SequenceOut.fifth THEN
			SequenceOut.fifth := vTemp;
		ELSIF SequenceIN.sixth = SequenceOut.seventh THEN
			SequenceOut.seventh := vTemp;
		ELSIF SequenceIN.sixth = SequenceOut.eight THEN
			SequenceOut.eight := vTemp;
		END_IF
	ELSIF SequenceIN.seventh <> SequenceOut.seventh THEN
			vTemp:= SequenceOut.seventh;
		SequenceOut.seventh := SequenceIN.seventh;
		(* Find the index where the same number is and write temp there
		but skip this position *)
		IF SequenceIN.seventh = SequenceOut.first THEN
			SequenceOut.first := vTemp;
		ELSIF SequenceIN.seventh = SequenceOut.second THEN
			SequenceOut.second := vTemp;
		ELSIF SequenceIN.seventh = SequenceOut.third THEN
			SequenceOut.third := vTemp;
		ELSIF SequenceIN.seventh = SequenceOut.fourth THEN
			SequenceOut.fourth := vTemp;
		ELSIF SequenceIN.seventh = SequenceOut.fifth THEN
			SequenceOut.fifth := vTemp;
		ELSIF SequenceIN.seventh = SequenceOut.sixth THEN
			SequenceOut.sixth := vTemp;
		ELSIF SequenceIN.seventh = SequenceOut.eight THEN
			SequenceOut.eight := vTemp;
		END_IF
	ELSIF SequenceIN.eight <> SequenceOut.eight THEN
			vTemp:= SequenceOut.eight;
		SequenceOut.eight := SequenceIN.eight;
		(* Find the index where the same number is and write temp there
		but skip this position *)
		IF SequenceIN.eight = SequenceOut.first THEN
			SequenceOut.first := vTemp;
		ELSIF SequenceIN.eight = SequenceOut.second THEN
			SequenceOut.second := vTemp;
		ELSIF SequenceIN.eight = SequenceOut.third THEN
			SequenceOut.third := vTemp;
		ELSIF SequenceIN.eight = SequenceOut.fourth THEN
			SequenceOut.fourth := vTemp;
		ELSIF SequenceIN.eight = SequenceOut.fifth THEN
			SequenceOut.fifth := vTemp;
		ELSIF SequenceIN.eight = SequenceOut.sixth THEN
			SequenceOut.sixth := vTemp;
		ELSIF SequenceIN.eight = SequenceOut.seventh THEN
			SequenceOut.seventh := vTemp;
		END_IF
	ELSE
		vTemp := 0;
	END_IF
ELSE
	vTemp:= 0;
	SequenceOut := SequenceIN;
END_IF;
          
END_FUNCTION_BLOCK

PROGRAM VJEZBA_PID
  VAR
    Kontroler : PID;
    vIzlazProcesa : REAL;
    Proces : REAL;
    Smetnja : REAL;
    vSP : REAL;
    vMan : BOOL;
    vRes : BOOL;
    IzlazPID : REAL;
    vKp : REAL;
    vTn : REAL;
    vTv : REAL;
    vManY : REAL;
    vOffSet : REAL;
  END_VAR

            (**)
vIzlazProcesa:=Proces+Smetnja+IzlazPID;

Kontroler(
	ACTUAL:= vIzlazProcesa, 
	SET_POINT:= vSP, 
	KP:= vKp, 
	TN:= vTn, 
	TV:= vTv, 
	Y_MANUAL:= vManY, 
	Y_OFFSET:= vOffSet, 
	Y_MIN:=1 , 
	Y_MAX:= 100, 
	MANUAL:=vMan , 
	RESET:= vRes, 
	Y=>IzlazPID , 
	LIMITS_ACTIVE=> , 
	OVERFLOW=> );
          
END_PROGRAM

PROGRAM VJEZBA0
  VAR
    Ventilator : MotorVentilator;  (* 10kV, 1 MW ELektromotor *)
    StartRequirements : BOOL;
    StopRequirements : BOOL;
    MotorStart : BOOL;
    MotorFail : BOOL;
    MotorDisablements : BOOL;
    iStartSWB : BOOL;
    iStartRemote : BOOL;
    StartPLC : BOOL;
    MotorStop : BOOL;
    iStopSWB : BOOL;
    iStopRemote : BOOL;
    StopPLC : BOOL;
    iMotor_CB_Closed : BOOL := TRUE;
    iMotor_CB_Earthed : BOOL := FALSE;
    MotorProtection : BOOL;
    Counter : INT := 0;
    iEMCY_Remote : BOOL := TRUE;
    iEMCY_SWB : BOOL := TRUE;
    EMCY_Group : BOOL;
    qLamp_Remote : BOOL;
    qLamp_SWB : BOOL;
    RHS : INT;
    StartTrig : R_TRIG;
    StartCount : INT;
    LampBlink05HZ : BOOL;
    MotorDelayStart : BOOL;
    ResetRHS : BOOL;
    LightBlinker05HZ : INT;
    RHSBlink : BOOL;
    StartCountBlink : BOOL;
    ResetButtonVisible : BOOL;
    Current : INT;
    StartDelay : TP;
  END_VAR

            (*
VJEŽBA 0: UPRAVLJANJE SREDNJENAPONSKIM NEREGULIRANIM
ELEKTROMOTORNIM POGONOM S DIREKTNIM UKLJUČIVANJEM
Cilj vježbe: Naučiti osnove programiranja programirljivih logičkih kontrolera (PLC-ova),
primijeniti PLC za automatizaciju tipičnog industrijskog postrojenja
Opis tehnološkog procesa:
Prozračivanje proizvodne hale obavlja se usisnim ventilatorom kojeg pogoni srednjenaponski (10kV, 1MW)
elektromotor. Elektromotor se pokreće direktnim upuštanjem i to prekidačem ugrađenim u sklopu SN razvodne
ploče.*)

MotorFail := Ventilator.iMotorFailOther OR Ventilator.iOvercurrentProtection OR Ventilator.iOverheatProtection;

Ventilator.qMotor := 		 StartRequirements
 						AND (MotorStart OR Ventilator.qMotor)
			   			AND NOT StopRequirements
			    		AND NOT MotorStop;

(*Sustav ventilacije je samo dio složenijeg proizvodnog procesa kojim upravlja PLC. Kako je većina uređaja pod
kontrolom PLCa niskonaponska, upravljački ormarić sa PLCom i popratnom opremom se nalazi u prostoriji sa
nisko naponskom razvodno-upravljačkom pločom.
U neposrednoj blizini motora je postavljena lokalna upravljačka konzola na kojoj su smještene tipkala, preklopke
i signalne sijalice kojima operater upravlja radom motora.*)

(*Motor može pokrenuti/zaustaviti (prema prioritetnom redu):
• operater komandama sa motornog polja ploče srednjeg napona,
• operater sa lokalne upravljačke konzole,
• operater iz udaljene komandne prostorije (eng. control room) pomoću SCADA sustava ili
• program PLC-a kada to zahtjeva tehnološki ciklus.*)

MotorStart := (Ventilator.iStart_Local OR iStartSWB OR iStartRemote OR StartPLC) AND NOT MotorDelayStart;
MotorStop := Ventilator.iStop_Local OR iStopSWB OR iStopRemote OR StopPLC;

(*Da bi se motor mogao pokrenuti, moraju za to biti ispunjeni preduvjeti poput:
• prekidač motora je u radnoj poziciji, spreman za zatvaranje,
• rastavljač za uzemljenje motora mora biti otvoren,
• niti jedna zaštita motora ne smije biti aktivna,
• glavno i pomoćno napajanje mora biti prisutno,
• niti jedno tipkalo za isklop u nuždi ("gljiva") nije aktivirano,
• proteklo je dovoljno vremena (vremenska zadrška) od posljednjeg starta itd.*)

StartRequirements := iMotor_CB_Closed AND NOT iMotor_CB_Earthed AND NOT MotorFail AND EMCY_Group;

IF iEMCY_Remote AND Ventilator.iEmcy_Stop AND iEMCY_SWB THEN
	EMCY_Group := TRUE;
ELSE
	EMCY_Group := FALSE;
	iMotor_CB_Closed := FALSE; (*TripCB*)
END_IF

IF Ventilator.iOvercurrentProtection THEN
	iMotor_CB_Closed := FALSE;
END_IF

(*Većina od ovih zahtjeva blokira pokretanje motora "ožičenom logikom". Osim ovih (osnovnih) uvjeta, postoje
dodatni uvjeti koji moraju, ovisno o mjestu i načinu upravljanja motorom, biti ispunjeni prije pokretanja motora:
• klapne na usisnoj grani ventilatora moraju biti zatvorene (manji udar na mrežu),
• ostali dijelovi sustava ventilacije moraju biti funkcionalni,
• pretpostavke za ekonomičan rad moraju biti ispunjene, itd.
Za potrebe laboratorijske vježbe će funkcionalnost sustava biti pojednostavljena, a broj U/I linija sveden na
minimum. Stoga će se koristiti samo signali čije su U/I linije PLCa označene punom linijom na slici 1.*)

(*Napomena: Isklop u nuždi mora biti izveden u "ožičenoj logici" i mora zaustaviti cijeli pogon ili samo jedan njegov dio
(zonu) neovisno o radu PLCa. Uglavnom se izvodi tako da prekida pomoćno napajanje sklopnika ili djeluje na ulaz za
otvaranje prekidača u svrhu dovođenja uređaja u beznaponsko stanje.*)
 
(*Kratak opis upravljačkog programa
Upravljački program PLCa mora osigurati jednostavno vođenje motora ventilatora sa lokalne upravljačke
konzole. Uz funkcije koje su date u opisu signalnih linija, program mora ispuniti i slijedeće zahtjeve:
1. motor se smije pokrenuti (zahtjev za start motora smije se poslati) samo ukoliko za to ispunjeni svi uvjeti
2. prebacivanjem kontrole motora sa lokalnog upravljanja (kontrole na MV ploči) na daljinsko upravljanje
(PLC) mora se održati status rada motora (ukoliko motor radi ne smije stati i obrnuto)
3. status motora i popratne opreme mora biti vidljiv na lokalnoj upravljačkoj. To se izvodi pomoću READY
signalne sijalice po slijedećoj shemi:
• ugašena, motor radi normalan rad motora
• ugašena, motor ne radi blokada aktivna u MV ploči (MV_SWBD_RDY_DI=0)
• trajno svijetli, motor ne radi motor spreman za start
• trajno svijetli, motor radi kontrola sa MV ploče (MV_SWBD_REM_DI=0)
• treptanje sporo (0.5Hz), ne radi vremenska zadrška zbog opetovanog starta
• treptanje srednje (1Hz), ne radi prorada zaštite tijekom rada motora ili neuspješan
start(zabilježen događaj)
• treptanje brzo (2Hz), ne radi isklop u nuždi aktivan.*)

Ventilator.qLamp_Local := Ventilator.qMotor AND NOT RHSBlink AND NOT StartCountBlink;
qLamp_Remote := Ventilator.qMotor AND NOT RHSBlink AND NOT StartCountBlink;
qLamp_SWB := Ventilator.qMotor AND NOT RHSBlink AND NOT StartCountBlink;

(*Da bi se poništilo zabilježeno alarmno stanje (ispad motora) i dobio trenutan status spremnosti motora za
rad potrebno je pritisnuti STOP tipku.*)

IF Ventilator.iStop_Local OR iStopRemote OR iStopSWB THEN
	Ventilator.iMotorFailOther := FALSE;
	Ventilator.iOvercurrentProtection := FALSE;
	Ventilator.iOverheatProtection := FALSE;
END_IF

(*4. kako bi se smanjila termička naprezanja motora, motor se može startati 3 puta na sat ako je hladan ili 2 puta
na sat, ako je topao. Motor je hladan ako ne radi jedan sat. Ovaj zahtjev se realizira po principu (15-30) tj.
hladan motor se može startati 15 minuta nakon prvog i potom 30 minuta nakon svakog slijedećeg starta.
Za potrebe vježbe je potrebno napraviti blokadu pokretanja motora 1 minutu nakon zadnjeg upuštanja.*)
StartDelay(IN:=Ventilator.iStart_Local OR iStartSWB OR iStartRemote OR StartPLC, PT:=T#15S , Q=>MotorDelayStart);
(*
5. Radi potreba održavanja, potrebno je realizirati brojač sati rada motora i broja upuštanja. Ukoliko je broj sati
rada veći od 5000 ili broj upuštanja veći od 300, READY sijalica mora svakih 5 s nakratko promijeniti svoje
stanje.*)
LightBlinker05HZ := LightBlinker05HZ+1;
IF LightBlinker05HZ >= 0 AND LightBlinker05HZ < 25 THEN
	LampBlink05HZ:=TRUE;
ELSIF LightBlinker05HZ >=25 AND LightBlinker05HZ <50 THEN
	LampBlink05HZ:=FALSE;
ELSIF LightBlinker05HZ >=50	THEN
	LightBlinker05HZ := 0;
END_IF

IF ResetRHS THEN
	StartCount:=0;
	RHS:=0;
END_IF

StartTrig(CLK:=Ventilator.iStart_Local OR iStartRemote OR iStartSWB OR StartPLC);
IF StartTrig.Q THEN
	StartCount := StartCount + 1;
END_IF
IF StartCount >5 THEN
	StartCountBlink := LampBlink05HZ;
ELSE
	StartCountBlink := FALSE;
END_IF

IF Ventilator.qMotor THEN
	RHS := RHS + 1;
	IF RHS >= 2000 THEN
		RHSBlink := LampBlink05HZ;
	ELSE
		RHSBlink := FALSE;
	END_IF
END_IF
ResetButtonVisible := StartCount > 3 OR RHS > 1500;

IF Ventilator.qMotor THEN
	Current := 30;
ELSE
	Current := 0;
END_IF
          
END_PROGRAM

PROGRAM VJEZBA1
  VAR
    RUCNO_AUTO : BOOL;
    START_TIPKA : BOOL;
    STOP_TIPKA : BOOL;
    LAMP_TEST : BOOL;
    LEVEL_H_HIGH : BOOL;
    LEVEL_HIGH : BOOL;
    LEVEL_LOW : BOOL;
    LEVEL_L_LOW : BOOL;
    MOTOR_READY : BOOL;
    PUMPA : MotorPump;
    Ready_Lampa : BOOL;
    Run_Lampa : BOOL;
    Alarm_Lampa : BOOL;
    H_High_Lampa : BOOL;
    High_Lampa : BOOL;
    Low_Lampa : BOOL;
    L_Low_Lampa : BOOL;
    START_AUTO : BOOL;
    STOP_AUTO : BOOL;
    Motor_Start : BOOL;
    WaterLevel : REAL := 280;
    Inflow : REAL := 0;
    OutFlow : REAL := 0;
    DiffPressDelay : Ton;
    SimulateRain : BOOL;
    AlarmCreator : LIMITALARM;
    Alarm_Level_Too_High : BOOL;
    Alarm_Level_Too_Low : BOOL;
    RHS : INT;
    BlinkingLight : BLINK;
    ServiceLight : BOOL;
    RHS_Reset : BOOL;
  END_VAR

            (*Kolektor otpadnih voda*)
(*Opis tehnološkog procesa:
Otpadne vode slivaju se u spremnik sabirnika otpadnih voda. Spremnik se nalazi na najnižoj točki teritorija sa
kojeg se vode prikupljalju. Prije ispuštanja u more prikupljena voda se prečišćava u pogonima gradskog
kolektora. Da bi se otpadne vode dopremile u kolektor potrebno ih je prebaciti u gradski kanalizacijski sustav. Za
savladavanje visinske razlike između spremnika i priključka na kanalizacijski sustav koristi se pumpa pokretana
trofaznim asinkronim motorom.
Opis crpne stanice:
Vizualizacija 1 prikazuje shematski prikaz stanice. Stanica se sastoji od crpke pokretane trofaznim asinkronim motorom,
četiri magnetska nivo sklopke za dojavljivanje razine otpadnih voda, lokalnog upravljačkog ormarića
(upravljačke konzole), PLCa i motorske grupe za pokretanje i zaštitu motora.
Svaka nivo sklopka se nalazi na zasebnoj razini, dva na gornjoj, a dva na donjoj razini spremnika, prema
slijedećem rasporedu :
• Level High-High (LEV_HH) – jako visoka razina vode
• Level High (LEV_HI) – visoka razina vode
• Level Low (LEV_LO) – niska razina vode
• Level Low–Low (LEV_LL) – jako niska razina vode
Sklopka visokog nivoa LEV_HI signalizira da je nivo otpadnih voda dosegnuo razinu na kojoj je potrebno
uključiti motor crpke radi pražnjenja spremnika. Spremnik se prazni dok sklopka LEV_LO ne signalizira da je
spremnik dovoljno ispražnjen tj. da je dosegnuta razina vode pri koje je potrebno zaustaviti pogon crpke. Ostale
dvije sklopke imaju dvostruku ulogu: alarmiranje i zaštitu od otkazivanja. Sklopka LEV_HH može biti aktivirana
ukoliko je sklopka LEV_HI neispravna (ili blokirana krupnim otpadnim materijalom. npr. granjem) pa crpka nije
proradila na pravom nivou ili je dotok (npr. oborinskih voda) veći od kapaciteta crpke pa prijeti opasnost od
izlijevanja otpadnih voda u more kroz prelijevni ventil. Sklopka LEV_LL predstavlja veoma nisku razinu
otpadnih voda pri kojem prijeti opasnost od oštećenja crpke zbog povlačenja krutog plutajućeg otpada ili zbog
“suhog rada”. *)

IF SimulateRain THEN
	Inflow := Inflow - 0.25;
END_IF;

WaterLevel := Inflow + OutFlow;

IF PUMPA.Running THEN
	OutFlow := Outflow + 0.5;
	IF WaterLevel >280 THEN
		WaterLevel := 280;
	END_IF
END_IF

IF WaterLevel <=-100 THEN
	LEVEL_H_HIGH := TRUE;
	Alarm_Level_Too_High:=TRUE;
ELSIF WaterLevel <= -90 THEN
	LEVEL_HIGH := TRUE;
ELSE
	LEVEL_HIGH:=FALSE;
	LEVEL_H_HIGH := FALSE;
	Alarm_Level_Too_High:=FALSE;
END_IF

IF WaterLevel >=0 THEN
	LEVEL_L_LOW := TRUE;
	Alarm_Level_Too_Low:=TRUE;
ELSIF WaterLevel >= -10 THEN
	LEVEL_LOW := TRUE;
ELSE
	LEVEL_LOW:=FALSE;
	LEVEL_L_LOW := FALSE;
	Alarm_Level_Too_Low:=FALSE;
END_IF

	
(*Crpka je opremljena i diferencijalni senzor tlaka (diferencijalnom tlačnom sklopkom ili presostatom). Sklopka
aktivira izlazni signal ukoliko je razlika razlika tlakova na ulaznij i izlaznoj cijevi crpke veća od podešenog praga.
Prag sklopke se postavlja tako da odgovara razlici ulaznog i izlaznog tlaka pri ispravnom radu crpke.
Nepostojanje takvog tlaka tj. nepostojanje signala tlačne sklopke predstavlja neispravan rad rad crpke pri kojem
se mora zaustaviti rad pogonskog motora, a detektirano stanje se mora prikazati alarmom.*)


	DiffPressDelay (IN:=WaterLevel >10 AND PUMPA.Running, PT:=T#5S); (*Tu mora dati alarm*)
	IF DiffPressDelay.q THEN
		PUMPA.DiffPress := TRUE;
	ELSE
		PUMPA.DiffPress := FALSE;	
	END_IF

(*Postoje dva režima rada crpna stanice: ručno i automatski. Način rada se odabire preklopkom koja se nalazi na
upravljačkoj konzoli.
Ručni režim rada:
Ručni režim rada koristi se u izvanrednim situacijama: prilikom puštanja u rad, servisnih radova ili zbog takvog
otkaza opreme da je automatski rad onemogućen. U režimu ručnog rada operater preuzima kontrolu nad
pokretanjem i zaustavljanjem motora crpke START/STOP tipkalima, neovisno o signalima nivo sklopki.
Aktivna je zaštita koja zaustavlja motor u slučaju nedovoljne razlike tlaka na crpki.
Automatski režim rada:
Automatski režim rada je normalan režim rada. Podizanjem nivoa otpadnih voda i proradom nivo sklopke
LEV_HI pokreće se crpka. Crpka se isključuje kada je dosegnut niski nivo u spremniku, odnosno kada proradi
sklopka LEV_LO. Redundantne sklopke LEV_HH i LEV_LL moraju pokrenuti odnosno zaustaviti motor crpke
neovisno o položajima sklopki LEV_HI i LEV_LO. Aktivna je zaštita koja zaustavlja motor u slučaju
nedovoljne razlike tlaka na crpki.*)

(*Zaštita crpke i pogonskog motora
Mehanizam crpke štiti se isključivanjem pogonskog motora kada je dostignuta vrlo niska razina u spremniku
LEV_LL i kada je razlika tlakova na ulaznoj i izlaznoj ispod dopuštenoga. Radni tlak crpka postiže 2 sekunde
nakon pokretanja motora.
Elektro motor crpke štiti se bimetalnom zaštitom u sklopu startera motora. Za očitavanje stanja startera motora
koristi se beznaponski kontakt koji je zatvoren ukoliko je motor spreman za pokretanje. Prorada zaštite, ispad
napajanja ili pokretanje motora otvorit će signalni kontakt. Za provjeru da li motor radi odnosno da li je sklopnik
motora uključen koristi se MOTOR RUNNING linija koju zatvaraju pomoćni kontakti sklopnika motora. Signal
MOT_RUN služi za pokretanje motora. Motor će raditi (sklopnik motora će biti uključen) dok je signal aktivan.*)

START_AUTO := RUCNO_AUTO AND (LEVEL_HIGH OR LEVEL_H_HIGH);
STOP_AUTO := RUCNO_AUTO AND (LEVEL_LOW OR LEVEL_L_LOW);

IF RUCNO_AUTO THEN
	Motor_Start := (START_AUTO OR Motor_Start) AND NOT PUMPA.DiffPress AND NOT STOP_AUTO;
ELSE
	Motor_Start := (START_TIPKA OR Motor_Start) AND NOT PUMPA.DiffPress AND NOT STOP_TIPKA;
END_IF
PUMPA.Running := Motor_Start;

MOTOR_READY := NOT PUMPA.Running AND NOT PUMPA.DiffPress AND NOT PUMPA.Fail;
Ready_Lampa := MOTOR_READY OR ServiceLight;
H_HIGH_LAMPA := LEVEL_H_HIGH;
HIGH_LAMPA := LEVEL_HIGH;
Run_Lampa := PUMPA.Running;
Low_Lampa := LEVEL_LOW;
L_LOW_LAMPA := LEVEL_L_LOW;
Alarm_Lampa := PUMPA.DiffPress OR PUMPA.Fail OR LEVEL_H_HIGH OR LEVEL_L_LOW;

IF Lamp_Test THEN
	Ready_Lampa := TRUE;
	H_HIGH_LAMPA := TRUE;
	HIGH_LAMPA := TRUE;
	Run_Lampa := TRUE;
	Low_Lampa := TRUE;
	L_LOW_LAMPA := TRUE;
	Alarm_Lampa := TRUE;
ELSE
	Ready_Lampa := FALSE;
	H_HIGH_LAMPA := FALSE;
	HIGH_LAMPA := FALSE;
	Run_Lampa := FALSE;
	Low_Lampa := FALSE;
	L_LOW_LAMPA := FALSE;
	Alarm_Lampa := FALSE;
END_IF

(*Upravljačka konzola
Za odabir načina rada, pokretanje i zaustavljanje motora crpke te očitanje statusa postrojenja operater koristi
upravljačku konzolu. Ona se sastoji od preklopke za odabir režima rada, start tipkala, stop tipkala, tipkala za
provjeru sijalica, te signalnih sijalica za dojave razine vode u spremniku, alarma i rada motora. Izgled upravljačke
konzole vidi se na dijelu “KONTROLNI PANEL” makete crpne stanice (slika 2.)
Na upravljačkoj konzoli nalazi se sedam signalnih sijalica pomoću kojih se može odrediti stanje pojedinih
dijelova crpne stanice. To su:
• READY sijalica - potvrda spremnosti crpke za pokretanje, zahtjev za servis
• RUN sijalica - signalizira da motor crpke radi
• ALARM sijalica - signalizira da li je došlo i do koje greške u radu crpke
• 4 sijalice - prikaz stanja nivo sklopki.*)

(*Alarmi
Alarmi dojavljuju opasna stanja. Alarm može biti:
• aktivan - opasna situacija još uvijek prisutna
• nepotvrđen - opasna situacija je prošla,
• potvrđen - operator je reagirao na nepotvrđen alarm, alarmno stanje se gasi,
• tihi – alarmna situacija je još uvijek aktivna, ali je potvrđena sa strane operatera. Prestankom uzroka
alarmne situacije, alarm se gasi.
Alarmi koje treba realizirati u okviru vježbe su dati u tablici 2. Kako zvučno alarmiranje (alarmna sirena) nije
ugrađena u pogon, tihi alarm nije potrebno realizirati. Alarmna situacija se potvrđuje tipkalom LAMP TEST.*)



(*Zbog nepovoljnih uvjeta u kojima radi crpka (potpuno uronjena u otpadnu vodu) potrebno je obaviti servisni
pregled svakih 100 sati rada. Upravljački program PLCa prati broj sati rada od zadnjeg pregleda i dostizanjem
servisnog intervala postavlja zahtjev za servis na upravljačkoj konzoli.*)
IF PUMPA.Running THEN
	RHS:=RHS+1;
	IF RHS > 1000 THEN
		BlinkingLight(ENABLE:=TRUE, TIMELOW:=T#2S, TIMEHIGH:=T#2S, OUT=>ServiceLight);
	END_IF
END_IF
IF RHS>1000 AND RHS_Reset THEN
	RHS:=0;
END_IF;
          
END_PROGRAM

FUNCTION_BLOCK Pump_Model
  VAR_INPUT
    OnCmd : BOOL;  (* Pump simulator will turn on when recieves ON signal and will shutoff when it recieves a OFF signal If SimTrip signal becomes true, pump will trip and cannot be started until signal goes false If SimFilterFail signal becomes true the pump will operate but the flowrate will start to slowly drop until zero *)
    OffCmd : BOOL;
    SimTrip : BOOL := FALSE;
    SimFilterFail : BOOL := FALSE;
    NoWater : BOOL := FALSE;  (* This tells the pump simulation that there is no more medium to pump so the flowmeter drops to 0 *)
    cfgFlowrate : REAL := 3000;
    cfgRampUpRate : REAL := 150;
    cfgRampDownRate : REAL := 150;
  END_VAR
  VAR_OUTPUT
    RunStatus : DINT;  (* 0 - Stopped, 1 - Running *)
    FlowmeterOut : REAL;  (* Cubic meters per hour *)
  END_VAR
  VAR
    PumpSR : SR;
    vPumpRunning : BOOL;
    Flowmeter : RAMP_REAL;
    vFlowmeterSP : REAL;
    vAscend : REAL;
    vDescend : REAL;
  END_VAR

            
PumpSR(SET1:= OnCmd AND NOT (OffCmd OR SimTrip OR RunStatus=1) , RESET:= (OffCmd OR SimTrip), Q1=>vPumpRunning );

RunStatus := BOOL_TO_DINT(vPumpRunning);

IF vPumpRunning AND NOT NoWater THEN
	vFlowmeterSP := BOOL_TO_REAL( NOT SimFilterFail) * cfgFlowrate;
	vAscend := cfgRampUpRate;
	vDescend := cfgRampDownRate;
ELSE
	vFlowmeterSP := 0;
	vAscend := 0;
	vDescend := 99999999;
END_IF


Flowmeter(
	IN:= vFlowmeterSP, 
	ASCEND:= vAscend,
	TIMEBASE:= T#500MS, 
	DESCEND:= vDescend, 
	OUT=> FlowmeterOut);
          
END_FUNCTION_BLOCK

FUNCTION Rand : DINT
  VAR_IN_OUT
    seed : ULINT;
  END_VAR
  VAR_INPUT
    lower : UINT;
    upper : UINT;
  END_VAR
  VAR
    range : UINT := ((upper - lower) + 1);
    interval : UINT := (c4 / range);
    preRand : UINT;
  END_VAR
  VAR CONSTANT
    c1 : UDINT := 1103515245;
    c2 : UINT := 12345;
    c3 : UDINT := 65536;
    c4 : UINT := 32768;
  END_VAR

            seed := seed * c1 + c2;
preRand := ULINT_TO_UINT((seed/c3) MOD c4);
IF interval > 0 THEN
	Rand := (preRand+lower*interval-1)/interval; 
ELSE
	Rand := preRand;
END_IF;
RETURN;


          
END_FUNCTION

PROGRAM PLC_PRG
  VAR
    Lamp : ARRAY[0..39, 0..7] OF BOOL;  (* Array for multiplying the Lamp object in the visualisation *)
    Row0 : LINT;  (* Row 0 of the Lamp array *)
    Row1 : LINT;  (* Row 1 of the Lamp array *)
    Row2 : LINT;  (* Row 2 of the Lamp array *)
    Row3 : LINT;  (* Row 3 of the Lamp array *)
    Row4 : LINT;  (* Row 4 of the Lamp array *)
    Row5 : LINT;  (* Row 5 of the Lamp array *)
    Row6 : LINT;  (* Row 6 of the Lamp array *)
    Row7 : LINT;  (* Row 7 of the Lamp array *)
    Timer : TON;
    vSequence : INT;  (* Sequence selector for the case machine *)
    Start : BOOL;  (* Starts the simulation *)
    Stop : BOOL;  (* Stops the simulation *)
    ScrollText : BOOL;  (* Starts the scrolling text simulation *)
    TempBuff0 : LINT;
    TempBuff1 : LINT;
    TempBuff2 : LINT;
    TempBuff3 : LINT;
    TempBuff4 : LINT;
    TempBuff5 : LINT;
    TempBuff6 : LINT;
    TempBuff7 : LINT;
    n : INT := 1;  (* Number of places to shift *)
  END_VAR

            (*Project Scrolling Text, Toni Kucic, Finland/Croatia, 16.6.2017*)

(*Letter S= 16#7f,16#7f,16#60,16#7f,16#7f,16#3,16#7f,16#7f  *)
(*Letter C= 16#7f,16#7f,16#60,16#60,16#60,16#60,16#7f,16#7f *)
(*Letter A= 16#7f,16#7f,16#63,16#63,16#7f,16#7f,16#63,16#63 *)
(*Letter D= 16#7c,16#7e,16#63,16#63,16#63,16#63,16#7e,16#7c *)
(*Letter A= 16#7f,16#7f,16#63,16#63,16#7f,16#7f,16#63,16#63 *)

(*First task was to create an LCD screen that lights up sequentially following the scheme:
" ", "S", "C", "A", "D", "A", "SCADA".
Each part of the sequence is 5sec long therefore the whole sequence is 35sec After that its repeated.
There is a Start and a Stop control button. In the sequence 6, the scrolling text funcionality is added
 to which we enter from the sequence 5 and by pressing ScrollText Button.
Future plan is to create a feeding system that will scroll the text in a string variable. 
As far as 18.6.2017 that hasn't been done on the PLC/using ST code.*)

IF STOP THEN
	vSequence:=0;
END_IF

CASE vSequence OF
	0: 	Timer(IN:=TRUE,PT:=T#1S);
		Row0:=16#0;
		Row1:=16#0;
		Row2:=16#0;
		Row3:=16#0;
		Row4:=16#0;
		Row5:=16#0;
		Row6:=16#0;
		Row7:=16#0;
		
		IF Start  AND NOT Stop AND Timer.Q THEN
			Timer(IN:=FALSE);
			vSequence:=1;
		END_IF
		
	1:	Timer(IN:=TRUE,PT:=T#5S);
		Row0:=16#7F;
		Row1:=16#7F;
		Row2:=16#60;
		Row3:=16#7F;
		Row4:=16#7F;
		Row5:=16#3;
		Row6:=16#7F;
		Row7:=16#7F;
		IF Timer.Q THEN
			Timer(IN:=FALSE);
			vSequence:=2;
		END_IF
		
	2: Timer(IN:=TRUE,PT:=T#5S);
		Row0:=16#7F7F;
		Row1:=16#7F7F;
		Row2:=16#6060;
		Row3:=16#7F60;
		Row4:=16#7F60;
		Row5:=16#360;
		Row6:=16#7F7F;
		Row7:=16#7F7F;
		IF Timer.Q THEN
			Timer(IN:=FALSE);
			vSequence:=3;
		END_IF
		
	3: Timer(IN:=TRUE,PT:=T#5S);
		Row0:=16#7F7F7F;
		Row1:=16#7F7F7F;
		Row2:=16#606063;
		Row3:=16#7F6063;
		Row4:=16#7F607F;
		Row5:=16#3607F;
		Row6:=16#7F7F63;
		Row7:=16#7F7F63;
		IF Timer.Q THEN
			Timer(IN:=FALSE);
			vSequence:=4;
		END_IF
		
	4: Timer(IN:=TRUE,PT:=T#5S);
		Row0:=16#7F7F7F7C;
		Row1:=16#7F7F7F7E;
		Row2:=16#60606363;
		Row3:=16#7F606363;
		Row4:=16#7F607F63;
		Row5:=16#3607F63;
		Row6:=16#7F7F637E;
		Row7:=16#7F7F637C;
		IF Timer.Q THEN
			Timer(IN:=FALSE);
			vSequence:=5;
		END_IF
		
	5: Timer(IN:=TRUE,PT:=T#5S);
		Row0:=16#7F7F7F7C7F;
		Row1:=16#7F7F7F7E7F;
		Row2:=16#6060636363;
		Row3:=16#7F60636363;
		Row4:=16#7F607F637F;
		Row5:=16#3607F637F;
		Row6:=16#7F7F637E63;
		Row7:=16#7F7F637C63;
		IF Timer.Q THEN (*When done, go back to state 0 and the sequence is repeating*)
			Timer(IN:=FALSE);
			vSequence:=0;
		ELSIF ScrollText THEN (*If the button scroll text is pressed the loop is broken and it goes to state 6, where it scrolls the text*)
			vSequence:=6;
		END_IF
	6: 
		Timer(IN:=NOT Timer.Q, PT:=T#0.25S);
		IF Timer.Q THEN
			TempBuff0.0 := Row0.39; (*Put last usable bit value to temporary buffer*)
			TempBuff1.0 := Row1.39;
			TempBuff2.0 := Row2.39;
			TempBuff3.0 := Row3.39;
			TempBuff4.0 := Row4.39;
			TempBuff5.0 := Row5.39;
			TempBuff6.0 := Row6.39;
			TempBuff7.0 := Row7.39;

			Row0:=SHL(Row0,n); (*Shift the data one bit to the left*)
			Row1:=SHL(Row1,n);
			Row2:=SHL(Row2,n);
			Row3:=SHL(Row3,n);
			Row4:=SHL(Row4,n);
			Row5:=SHL(Row5,n);
			Row6:=SHL(Row6,n);
			Row7:=SHL(Row7,n);

			Row0.0:=TempBuff0.0; (*The last bit of data that has moved gets put back to the beggining*)
			Row1.0:=TempBuff1.0;
			Row2.0:=TempBuff2.0;
			Row3.0:=TempBuff3.0;
			Row4.0:=TempBuff4.0;
			Row5.0:=TempBuff5.0;
			Row6.0:=TempBuff6.0;
			Row7.0:=TempBuff7.0;
		END_IF;
END_CASE

(*Lamp system 40x8*)
Lamp[0, 0]:=Row0.39;
Lamp[0, 1]:=Row1.39;
Lamp[0, 2]:=Row2.39;
Lamp[0, 3]:=Row3.39;
Lamp[0, 4]:=Row4.39;
Lamp[0, 5]:=Row5.39;
Lamp[0, 6]:=Row6.39;
Lamp[0, 7]:=Row7.39;
Lamp[1, 0]:=Row0.38;
Lamp[1, 1]:=Row1.38;
Lamp[1, 2]:=Row2.38;
Lamp[1, 3]:=Row3.38;
Lamp[1, 4]:=Row4.38;
Lamp[1, 5]:=Row5.38;
Lamp[1, 6]:=Row6.38;
Lamp[1, 7]:=Row7.38;
Lamp[2, 0]:=Row0.37;
Lamp[2, 1]:=Row1.37;
Lamp[2, 2]:=Row2.37;
Lamp[2, 3]:=Row3.37;
Lamp[2, 4]:=Row4.37;
Lamp[2, 5]:=Row5.37;
Lamp[2, 6]:=Row6.37;
Lamp[2, 7]:=Row7.37;
Lamp[3, 0]:=Row0.36;
Lamp[3, 1]:=Row1.36;
Lamp[3, 2]:=Row2.36;
Lamp[3, 3]:=Row3.36;
Lamp[3, 4]:=Row4.36;
Lamp[3, 5]:=Row5.36;
Lamp[3, 6]:=Row6.36;
Lamp[3, 7]:=Row7.36;
Lamp[4, 0]:=Row0.35;
Lamp[4, 1]:=Row1.35;
Lamp[4, 2]:=Row2.35;
Lamp[4, 3]:=Row3.35;
Lamp[4, 4]:=Row4.35;
Lamp[4, 5]:=Row5.35;
Lamp[4, 6]:=Row6.35;
Lamp[4, 7]:=Row7.35;
Lamp[5, 0]:=Row0.34;
Lamp[5, 1]:=Row1.34;
Lamp[5, 2]:=Row2.34;
Lamp[5, 3]:=Row3.34;
Lamp[5, 4]:=Row4.34;
Lamp[5, 5]:=Row5.34;
Lamp[5, 6]:=Row6.34;
Lamp[5, 7]:=Row7.34;
Lamp[6, 0]:=Row0.33;
Lamp[6, 1]:=Row1.33;
Lamp[6, 2]:=Row2.33;
Lamp[6, 3]:=Row3.33;
Lamp[6, 4]:=Row4.33;
Lamp[6, 5]:=Row5.33;
Lamp[6, 6]:=Row6.33;
Lamp[6, 7]:=Row7.33;
Lamp[7, 0]:=Row0.32;
Lamp[7, 1]:=Row1.32;
Lamp[7, 2]:=Row2.32;
Lamp[7, 3]:=Row3.32;
Lamp[7, 4]:=Row4.32;
Lamp[7, 5]:=Row5.32;
Lamp[7, 6]:=Row6.32;
Lamp[7, 7]:=Row7.32;
Lamp[8, 0]:=Row0.31;
Lamp[8, 1]:=Row1.31;
Lamp[8, 2]:=Row2.31;
Lamp[8, 3]:=Row3.31;
Lamp[8, 4]:=Row4.31;
Lamp[8, 5]:=Row5.31;
Lamp[8, 6]:=Row6.31;
Lamp[8, 7]:=Row7.31;
Lamp[9, 0]:=Row0.30;
Lamp[9, 1]:=Row1.30;
Lamp[9, 2]:=Row2.30;
Lamp[9, 3]:=Row3.30;
Lamp[9, 4]:=Row4.30;
Lamp[9, 5]:=Row5.30;
Lamp[9, 6]:=Row6.30;
Lamp[9, 7]:=Row7.30;
Lamp[10, 0]:=Row0.29;
Lamp[10, 1]:=Row1.29;
Lamp[10, 2]:=Row2.29;
Lamp[10, 3]:=Row3.29;
Lamp[10, 4]:=Row4.29;
Lamp[10, 5]:=Row5.29;
Lamp[10, 6]:=Row6.29;
Lamp[10, 7]:=Row7.29;
Lamp[11, 0]:=Row0.28;
Lamp[11, 1]:=Row1.28;
Lamp[11, 2]:=Row2.28;
Lamp[11, 3]:=Row3.28;
Lamp[11, 4]:=Row4.28;
Lamp[11, 5]:=Row5.28;
Lamp[11, 6]:=Row6.28;
Lamp[11, 7]:=Row7.28;
Lamp[12, 0]:=Row0.27;
Lamp[12, 1]:=Row1.27;
Lamp[12, 2]:=Row2.27;
Lamp[12, 3]:=Row3.27;
Lamp[12, 4]:=Row4.27;
Lamp[12, 5]:=Row5.27;
Lamp[12, 6]:=Row6.27;
Lamp[12, 7]:=Row7.27;
Lamp[13, 0]:=Row0.26;
Lamp[13, 1]:=Row1.26;
Lamp[13, 2]:=Row2.26;
Lamp[13, 3]:=Row3.26;
Lamp[13, 4]:=Row4.26;
Lamp[13, 5]:=Row5.26;
Lamp[13, 6]:=Row6.26;
Lamp[13, 7]:=Row7.26;
Lamp[14, 0]:=Row0.25;
Lamp[14, 1]:=Row1.25;
Lamp[14, 2]:=Row2.25;
Lamp[14, 3]:=Row3.25;
Lamp[14, 4]:=Row4.25;
Lamp[14, 5]:=Row5.25;
Lamp[14, 6]:=Row6.25;
Lamp[14, 7]:=Row7.25;
Lamp[15, 0]:=Row0.24;
Lamp[15, 1]:=Row1.24;
Lamp[15, 2]:=Row2.24;
Lamp[15, 3]:=Row3.24;
Lamp[15, 4]:=Row4.24;
Lamp[15, 5]:=Row5.24;
Lamp[15, 6]:=Row6.24;
Lamp[15, 7]:=Row7.24;
Lamp[16, 0]:=Row0.23;
Lamp[16, 1]:=Row1.23;
Lamp[16, 2]:=Row2.23;
Lamp[16, 3]:=Row3.23;
Lamp[16, 4]:=Row4.23;
Lamp[16, 5]:=Row5.23;
Lamp[16, 6]:=Row6.23;
Lamp[16, 7]:=Row7.23;
Lamp[17, 0]:=Row0.22;
Lamp[17, 1]:=Row1.22;
Lamp[17, 2]:=Row2.22;
Lamp[17, 3]:=Row3.22;
Lamp[17, 4]:=Row4.22;
Lamp[17, 5]:=Row5.22;
Lamp[17, 6]:=Row6.22;
Lamp[17, 7]:=Row7.22;
Lamp[18, 0]:=Row0.21;
Lamp[18, 1]:=Row1.21;
Lamp[18, 2]:=Row2.21;
Lamp[18, 3]:=Row3.21;
Lamp[18, 4]:=Row4.21;
Lamp[18, 5]:=Row5.21;
Lamp[18, 6]:=Row6.21;
Lamp[18, 7]:=Row7.21;
Lamp[19, 0]:=Row0.20;
Lamp[19, 1]:=Row1.20;
Lamp[19, 2]:=Row2.20;
Lamp[19, 3]:=Row3.20;
Lamp[19, 4]:=Row4.20;
Lamp[19, 5]:=Row5.20;
Lamp[19, 6]:=Row6.20;
Lamp[19, 7]:=Row7.20;
Lamp[20, 0]:=Row0.19;
Lamp[20, 1]:=Row1.19;
Lamp[20, 2]:=Row2.19;
Lamp[20, 3]:=Row3.19;
Lamp[20, 4]:=Row4.19;
Lamp[20, 5]:=Row5.19;
Lamp[20, 6]:=Row6.19;
Lamp[20, 7]:=Row7.19;
Lamp[21, 0]:=Row0.18;
Lamp[21, 1]:=Row1.18;
Lamp[21, 2]:=Row2.18;
Lamp[21, 3]:=Row3.18;
Lamp[21, 4]:=Row4.18;
Lamp[21, 5]:=Row5.18;
Lamp[21, 6]:=Row6.18;
Lamp[21, 7]:=Row7.18;
Lamp[22, 0]:=Row0.17;
Lamp[22, 1]:=Row1.17;
Lamp[22, 2]:=Row2.17;
Lamp[22, 3]:=Row3.17;
Lamp[22, 4]:=Row4.17;
Lamp[22, 5]:=Row5.17;
Lamp[22, 6]:=Row6.17;
Lamp[22, 7]:=Row7.17;
Lamp[23, 0]:=Row0.16;
Lamp[23, 1]:=Row1.16;
Lamp[23, 2]:=Row2.16;
Lamp[23, 3]:=Row3.16;
Lamp[23, 4]:=Row4.16;
Lamp[23, 5]:=Row5.16;
Lamp[23, 6]:=Row6.16;
Lamp[23, 7]:=Row7.16;
Lamp[24, 0]:=Row0.16;
Lamp[24, 1]:=Row1.15;
Lamp[24, 2]:=Row2.15;
Lamp[24, 3]:=Row3.15;
Lamp[24, 4]:=Row4.15;
Lamp[24, 5]:=Row5.15;
Lamp[24, 6]:=Row6.15;
Lamp[24, 7]:=Row7.15;
Lamp[25, 0]:=Row0.14;
Lamp[25, 1]:=Row1.14;
Lamp[25, 2]:=Row2.14;
Lamp[25, 3]:=Row3.14;
Lamp[25, 4]:=Row4.14;
Lamp[25, 5]:=Row5.14;
Lamp[25, 6]:=Row6.14;
Lamp[25, 7]:=Row7.14;
Lamp[26, 0]:=Row0.13;
Lamp[26, 1]:=Row1.13;
Lamp[26, 2]:=Row2.13;
Lamp[26, 3]:=Row3.13;
Lamp[26, 4]:=Row4.13;
Lamp[26, 5]:=Row5.13;
Lamp[26, 6]:=Row6.13;
Lamp[26, 7]:=Row7.13;
Lamp[27, 0]:=Row0.12;
Lamp[27, 1]:=Row1.12;
Lamp[27, 2]:=Row2.12;
Lamp[27, 3]:=Row3.12;
Lamp[27, 4]:=Row4.12;
Lamp[27, 5]:=Row5.12;
Lamp[27, 6]:=Row6.12;
Lamp[27, 7]:=Row7.12;
Lamp[28, 0]:=Row0.11;
Lamp[28, 1]:=Row1.11;
Lamp[28, 2]:=Row2.11;
Lamp[28, 3]:=Row3.11;
Lamp[28, 4]:=Row4.11;
Lamp[28, 5]:=Row5.11;
Lamp[28, 6]:=Row6.11;
Lamp[28, 7]:=Row7.11;
Lamp[29, 0]:=Row0.10;
Lamp[29, 1]:=Row1.10;
Lamp[29, 2]:=Row2.10;
Lamp[29, 3]:=Row3.10;
Lamp[29, 4]:=Row4.10;
Lamp[29, 5]:=Row5.10;
Lamp[29, 6]:=Row6.10;
Lamp[29, 7]:=Row7.10;
Lamp[30, 0]:=Row0.9;
Lamp[30, 1]:=Row1.9;
Lamp[30, 2]:=Row2.9;
Lamp[30, 3]:=Row3.9;
Lamp[30, 4]:=Row4.9;
Lamp[30, 5]:=Row5.9;
Lamp[30, 6]:=Row6.9;
Lamp[30, 7]:=Row7.9;
Lamp[31, 0]:=Row0.8;
Lamp[31, 1]:=Row1.8;
Lamp[31, 2]:=Row2.8;
Lamp[31, 3]:=Row3.8;
Lamp[31, 4]:=Row4.8;
Lamp[31, 5]:=Row5.8;
Lamp[31, 6]:=Row6.8;
Lamp[31, 7]:=Row7.8;
Lamp[32, 0]:=Row0.7;
Lamp[32, 1]:=Row1.7;
Lamp[32, 2]:=Row2.7;
Lamp[32, 3]:=Row3.7;
Lamp[32, 4]:=Row4.7;
Lamp[32, 5]:=Row5.7;
Lamp[32, 6]:=Row6.7;
Lamp[32, 7]:=Row7.7;
Lamp[33, 0]:=Row0.6;
Lamp[33, 1]:=Row1.6;
Lamp[33, 2]:=Row2.6;
Lamp[33, 3]:=Row3.6;
Lamp[33, 4]:=Row4.6;
Lamp[33, 5]:=Row5.6;
Lamp[33, 6]:=Row6.6;
Lamp[33, 7]:=Row7.6;
Lamp[34, 0]:=Row0.5;
Lamp[34, 1]:=Row1.5;
Lamp[34, 2]:=Row2.5;
Lamp[34, 3]:=Row3.5;
Lamp[34, 4]:=Row4.5;
Lamp[34, 5]:=Row5.5;
Lamp[34, 6]:=Row6.5;
Lamp[34, 7]:=Row7.5;
Lamp[35, 0]:=Row0.4;
Lamp[35, 1]:=Row1.4;
Lamp[35, 2]:=Row2.4;
Lamp[35, 3]:=Row3.4;
Lamp[35, 4]:=Row4.4;
Lamp[35, 5]:=Row5.4;
Lamp[35, 6]:=Row6.4;
Lamp[35, 7]:=Row7.4;
Lamp[36, 0]:=Row0.3;
Lamp[36, 1]:=Row1.3;
Lamp[36, 2]:=Row2.3;
Lamp[36, 3]:=Row3.3;
Lamp[36, 4]:=Row4.3;
Lamp[36, 5]:=Row5.3;
Lamp[36, 6]:=Row6.3;
Lamp[36, 7]:=Row7.3;
Lamp[37, 0]:=Row0.2;
Lamp[37, 1]:=Row1.2;
Lamp[37, 2]:=Row2.2;
Lamp[37, 3]:=Row3.2;
Lamp[37, 4]:=Row4.2;
Lamp[37, 5]:=Row5.2;
Lamp[37, 6]:=Row6.2;
Lamp[37, 7]:=Row7.2;
Lamp[38, 0]:=Row0.1;
Lamp[38, 1]:=Row1.1;
Lamp[38, 2]:=Row2.1;
Lamp[38, 3]:=Row3.1;
Lamp[38, 4]:=Row4.1;
Lamp[38, 5]:=Row5.1;
Lamp[38, 6]:=Row6.1;
Lamp[38, 7]:=Row7.1;
Lamp[39, 0]:=Row0.0;
Lamp[39, 1]:=Row1.0;
Lamp[39, 2]:=Row2.0;
Lamp[39, 3]:=Row3.0;
Lamp[39, 4]:=Row4.0;
Lamp[39, 5]:=Row5.0;
Lamp[39, 6]:=Row6.0;
Lamp[39, 7]:=Row7.0;


          
END_PROGRAM

FUNCTION_BLOCK ShiftArray
  VAR_IN_OUT
    DataArray : ARRAY[0..31] OF DINT;  (* 32 bit array of dints that will be shifted *)
  END_VAR
  VAR_INPUT
    ShiftLeft : BOOL;  (* Shifting left by one index. Trigger based *)
    ShiftRight : BOOL;  (* Shifting right by one index. Trigger based *)
    Value : DINT;  (* Value to be inserted *)
  END_VAR
  VAR
    ShiftLeftTrig : R_TRIG;
    ShiftRightTrig : R_TRIG;
    i : INT;
  END_VAR

            ShiftLeftTrig(CLK:=ShiftLeft);
ShiftRightTrig(CLK:=ShiftRight);

IF ShiftRightTrig.Q THEN
	FOR i := 31 TO 1 BY -1 DO
		DataArray[i]:= DataArray[i-1];
	END_FOR;
	DataArray[0]:= Value;
ELSIF ShiftLeftTrig.Q THEN
	FOR i := 0 TO 30 BY 1 DO
		DataArray[i]:= DataArray[i+1];
	END_FOR;
	DataArray[31]:= Value;
END_IF
          
END_FUNCTION_BLOCK

PROGRAM ShiftPOU
  VAR
    ShiftArray : ShiftArray;
    SomeArray : ARRAY[0..31] OF DINT;
    vShiftLeft : BOOL;
    vShiftRight : BOOL;
    vValue : DINT;
  END_VAR

            
ShiftArray(
	DataArray:= SomeArray,
	ShiftLeft:= vShiftLeft,
	ShiftRight:= vShiftRight,
	Value := vValue);
	
	
          
END_PROGRAM

PROGRAM POU
  VAR
    vStartGame : BOOL;
    PushButtonStart : INT;
    Candidate1Lamp : INT;
    Candidate2Lamp : INT;
    Candidate3Lamp : INT;
    PushButtonReset : INT;
    TimeOut : INT;
    GameTime : INT;
    IN : INT;
    PT : INT;
  END_VAR

            // vStartGame := (Task02GVL.PushButtonStart OR vStartGame)
// 		 AND NOT Task02GVL.Candidate1Lamp
// 		 AND NOT Task02GVL.Candidate2Lamp
// 		 AND NOT Task02GVL.Candidate3Lamp
// 		 AND NOT Task02GVL.PushButtonReset;
// 
// TimeOut(IN:=vStartGame,PT:=Task02GVL.GameTime);
// Task02GVL.Buzzer := TimeOut.Q;
// 
// IF vStartGame THEN
// Task02GVL.Candidate1Lamp := (Task02GVL.Candidate1PushButton OR Task02GVL.Candidate1Lamp) AND NOT TimeOut.Q;
// Task02GVL.Candidate2Lamp := (Task02GVL.Candidate2PushButton OR Task02GVL.Candidate2Lamp) AND NOT TimeOut.Q;
// Task02GVL.Candidate3Lamp := (Task02GVL.Candidate3PushButton OR Task02GVL.Candidate3Lamp) AND NOT TimeOut.Q;
// END_IF;
// 
// IF Task02GVL.Candidate1Lamp THEN
// 	Task02GVL.Candidate2Lamp:=FALSE;
// 	Task02GVL.Candidate3Lamp:=FALSE;
// ELSIF Task02GVL.Candidate2Lamp THEN
// 	Task02GVL.Candidate3Lamp:=FALSE;
// 	Task02GVL.Candidate1Lamp:=FALSE;
// ELSIF Task02GVL.Candidate3Lamp THEN
// 	Task02GVL.Candidate2Lamp:=FALSE;
// 	Task02GVL.Candidate1Lamp:=FALSE;	
// END_IF
// 
// IF Task02GVL.PushButtonReset THEN
// 	Task02GVL.Candidate1Lamp:=FALSE;
// 	Task02GVL.Candidate2Lamp:=FALSE;
// 	Task02GVL.Candidate3Lamp:=FALSE;
// END_IF
// 

          
END_PROGRAM

PROGRAM Zadatak4
  VAR
    M3 : BOOL;
    Start_Desno : BOOL;
    Start_Lijevo : BOOL;
    STOP : BOOL;
    SklopkaPreopterecenja : BOOL;
    M3_Lijevo : BOOL;
    M3_Desno : BOOL;
    Cooling : TOF;
    StreliceLijevoInv : BOOL;
    StreliceDesnoInv : BOOL;
  END_VAR

            (*Zadatak 4.
Promena smera obrtanja trofaznog asinhronog motora izvodi se promenom redosleda faza napona
napajanja motora. Upravljanje motorom izvodi se tasterima "START-DESNO", "START-LEVO" i "STOP".
Motor se sem toga štiti i od preopterećenja motornom zaštitnom sklopkom.
Razraditi rešenje kašnjenja sa PLC kontrolerom.*)

M3_Lijevo:=(M3_Lijevo OR Start_Lijevo) AND NOT M3_Desno AND NOT STOP AND NOT SklopkaPreopterecenja AND NOT Cooling.Q;
M3_Desno:=(M3_Desno OR Start_Desno) AND NOT M3_Lijevo AND NOT STOP AND NOT SklopkaPreopterecenja AND NOT Cooling.Q;

M3:= M3_Lijevo OR M3_Desno; (*Ovo je samo simulirani motor jer nemamo pravi*)
Cooling(IN:=Stop, PT:=T#5S);
StreliceLijevoInv:=M3_Desno OR (NOT M3_Desno AND NOT M3_Lijevo);
StreliceDesnoInv:=M3_Lijevo OR (NOT M3_Desno AND NOT M3_Lijevo);

          
END_PROGRAM

PROGRAM Zadatak5
  VAR
    Lamp : ARRAY[0..39, 0..7] OF BOOL;
    dword0 : LINT;
    dword1 : LINT;
    dword2 : LINT;
    dword3 : LINT;
    dword4 : LINT;
    dword5 : LINT;
    dword6 : LINT;
    dword7 : LINT;
    Timer : TON;
    vSequence : INT;
    Start : BOOL;
    STOP : BOOL;
  END_VAR

            (*Slovo S= 0x7f,0x7f,0x60,0x7f,0x7f,0x3,0x7f,0x7f  *)
(*Slovo C= 0x7f,0x7f,0x60,0x60,0x60,0x60,0x7f,0x7f  *)
(*Slovo A= 0x7f,0x7f,0x63,0x63,0x7f,0x7f,0x63,0x63  *)
(*Slovo D= 0x7c,0x7e,0x63,0x63,0x63,0x63,0x7e,0x7c  *)
(*Slovo A= 0x7f,0x7f,0x63,0x63,0x7f,0x7f,0x63,0x63 *)

(*Svijetleća reklama pali se sekvencijalno po slijedećoj šemi:
" ", "S", "C", "A", "D", "A", "SCADA".
Trajanje svakog dijela sekvence traje pet sekundi, odnosno ukupno trideset pet sekundi, poslije čega se
sekvenca automatski ponavlja. Komande za upravljanje svijetlećom reklamom ostvaruju se komandnim tasterima
"START" i "STOP". Paljenje segmenata svijetleće reklame izvedeno je relejnim kontaktima.
Razraditi prijedlog za realizaciju datog upravljačkog zadatka primjenom PLC uređaja.*)

IF STOP THEN
	vSequence:=0;
END_IF

CASE vSequence OF
	0: 	Timer(IN:=TRUE,PT:=T#1S);
		dword0:=16#0;
		dword1:=16#0;
		dword2:=16#0;
		dword3:=16#0;
		dword4:=16#0;
		dword5:=16#0;
		dword6:=16#0;
		dword7:=16#0;
		
		IF Start  AND NOT Stop AND Timer.Q THEN
			Timer(IN:=FALSE);
			vSequence:=1;
		END_IF
		
	1:	Timer(IN:=TRUE,PT:=T#5S);
		dword0:=16#7F;
		dword1:=16#7F;
		dword2:=16#60;
		dword3:=16#7F;
		dword4:=16#7F;
		dword5:=16#3;
		dword6:=16#7F;
		dword7:=16#7F;
		IF Timer.Q THEN
			Timer(IN:=FALSE);
			vSequence:=2;
		END_IF
		
	2: Timer(IN:=TRUE,PT:=T#5S);
		dword0:=16#7F7F;
		dword1:=16#7F7F;
		dword2:=16#6060;
		dword3:=16#7F60;
		dword4:=16#7F60;
		dword5:=16#360;
		dword6:=16#7F7F;
		dword7:=16#7F7F;
		IF Timer.Q THEN
			Timer(IN:=FALSE);
			vSequence:=3;
		END_IF
		
	3: Timer(IN:=TRUE,PT:=T#5S);
		dword0:=16#7F7F7F;
		dword1:=16#7F7F7F;
		dword2:=16#606063;
		dword3:=16#7F6063;
		dword4:=16#7F607F;
		dword5:=16#3607F;
		dword6:=16#7F7F63;
		dword7:=16#7F7F63;
		IF Timer.Q THEN
			Timer(IN:=FALSE);
			vSequence:=4;
		END_IF
		
	4: Timer(IN:=TRUE,PT:=T#5S);
		dword0:=16#7F7F7F7C;
		dword1:=16#7F7F7F7E;
		dword2:=16#60606363;
		dword3:=16#7F606363;
		dword4:=16#7F607F63;
		dword5:=16#3607F63;
		dword6:=16#7F7F637E;
		dword7:=16#7F7F637C;
		IF Timer.Q THEN
			Timer(IN:=FALSE);
			vSequence:=5;
		END_IF
		
	5: Timer(IN:=TRUE,PT:=T#5S);
		dword0:=16#7F7F7F7C7F;
		dword1:=16#7F7F7F7E7F;
		dword2:=16#6060636363;
		dword3:=16#7F60636363;
		dword4:=16#7F607F637F;
		dword5:=16#3607F637F;
		dword6:=16#7F7F637E63;
		dword7:=16#7F7F637C63;
		IF Timer.Q THEN
			Timer(IN:=FALSE);
			vSequence:=0;
		END_IF
END_CASE

(*Lamp system 40x7*)
Lamp[0, 0]:=dword0.39;
Lamp[0, 1]:=dword1.39;
Lamp[0, 2]:=dword2.39;
Lamp[0, 3]:=dword3.39;
Lamp[0, 4]:=dword4.39;
Lamp[0, 5]:=dword5.39;
Lamp[0, 6]:=dword6.39;
Lamp[0, 7]:=dword7.39;
Lamp[1, 0]:=dword0.38;
Lamp[1, 1]:=dword1.38;
Lamp[1, 2]:=dword2.38;
Lamp[1, 3]:=dword3.38;
Lamp[1, 4]:=dword4.38;
Lamp[1, 5]:=dword5.38;
Lamp[1, 6]:=dword6.38;
Lamp[1, 7]:=dword7.38;
Lamp[2, 0]:=dword0.37;
Lamp[2, 1]:=dword1.37;
Lamp[2, 2]:=dword2.37;
Lamp[2, 3]:=dword3.37;
Lamp[2, 4]:=dword4.37;
Lamp[2, 5]:=dword5.37;
Lamp[2, 6]:=dword6.37;
Lamp[2, 7]:=dword7.37;
Lamp[3, 0]:=dword0.36;
Lamp[3, 1]:=dword1.36;
Lamp[3, 2]:=dword2.36;
Lamp[3, 3]:=dword3.36;
Lamp[3, 4]:=dword4.36;
Lamp[3, 5]:=dword5.36;
Lamp[3, 6]:=dword6.36;
Lamp[3, 7]:=dword7.36;
Lamp[4, 0]:=dword0.35;
Lamp[4, 1]:=dword1.35;
Lamp[4, 2]:=dword2.35;
Lamp[4, 3]:=dword3.35;
Lamp[4, 4]:=dword4.35;
Lamp[4, 5]:=dword5.35;
Lamp[4, 6]:=dword6.35;
Lamp[4, 7]:=dword7.35;
Lamp[5, 0]:=dword0.34;
Lamp[5, 1]:=dword1.34;
Lamp[5, 2]:=dword2.34;
Lamp[5, 3]:=dword3.34;
Lamp[5, 4]:=dword4.34;
Lamp[5, 5]:=dword5.34;
Lamp[5, 6]:=dword6.34;
Lamp[5, 7]:=dword7.34;
Lamp[6, 0]:=dword0.33;
Lamp[6, 1]:=dword1.33;
Lamp[6, 2]:=dword2.33;
Lamp[6, 3]:=dword3.33;
Lamp[6, 4]:=dword4.33;
Lamp[6, 5]:=dword5.33;
Lamp[6, 6]:=dword6.33;
Lamp[6, 7]:=dword7.33;
Lamp[7, 0]:=dword0.32;
Lamp[7, 1]:=dword1.32;
Lamp[7, 2]:=dword2.32;
Lamp[7, 3]:=dword3.32;
Lamp[7, 4]:=dword4.32;
Lamp[7, 5]:=dword5.32;
Lamp[7, 6]:=dword6.32;
Lamp[7, 7]:=dword7.32;
Lamp[8, 0]:=dword0.31;
Lamp[8, 1]:=dword1.31;
Lamp[8, 2]:=dword2.31;
Lamp[8, 3]:=dword3.31;
Lamp[8, 4]:=dword4.31;
Lamp[8, 5]:=dword5.31;
Lamp[8, 6]:=dword6.31;
Lamp[8, 7]:=dword7.31;
Lamp[9, 0]:=dword0.30;
Lamp[9, 1]:=dword1.30;
Lamp[9, 2]:=dword2.30;
Lamp[9, 3]:=dword3.30;
Lamp[9, 4]:=dword4.30;
Lamp[9, 5]:=dword5.30;
Lamp[9, 6]:=dword6.30;
Lamp[9, 7]:=dword7.30;
Lamp[10, 0]:=dword0.29;
Lamp[10, 1]:=dword1.29;
Lamp[10, 2]:=dword2.29;
Lamp[10, 3]:=dword3.29;
Lamp[10, 4]:=dword4.29;
Lamp[10, 5]:=dword5.29;
Lamp[10, 6]:=dword6.29;
Lamp[10, 7]:=dword7.29;
Lamp[11, 0]:=dword0.28;
Lamp[11, 1]:=dword1.28;
Lamp[11, 2]:=dword2.28;
Lamp[11, 3]:=dword3.28;
Lamp[11, 4]:=dword4.28;
Lamp[11, 5]:=dword5.28;
Lamp[11, 6]:=dword6.28;
Lamp[11, 7]:=dword7.28;
Lamp[12, 0]:=dword0.27;
Lamp[12, 1]:=dword1.27;
Lamp[12, 2]:=dword2.27;
Lamp[12, 3]:=dword3.27;
Lamp[12, 4]:=dword4.27;
Lamp[12, 5]:=dword5.27;
Lamp[12, 6]:=dword6.27;
Lamp[12, 7]:=dword7.27;
Lamp[13, 0]:=dword0.26;
Lamp[13, 1]:=dword1.26;
Lamp[13, 2]:=dword2.26;
Lamp[13, 3]:=dword3.26;
Lamp[13, 4]:=dword4.26;
Lamp[13, 5]:=dword5.26;
Lamp[13, 6]:=dword6.26;
Lamp[13, 7]:=dword7.26;
Lamp[14, 0]:=dword0.25;
Lamp[14, 1]:=dword1.25;
Lamp[14, 2]:=dword2.25;
Lamp[14, 3]:=dword3.25;
Lamp[14, 4]:=dword4.25;
Lamp[14, 5]:=dword5.25;
Lamp[14, 6]:=dword6.25;
Lamp[14, 7]:=dword7.25;
Lamp[15, 0]:=dword0.24;
Lamp[15, 1]:=dword1.24;
Lamp[15, 2]:=dword2.24;
Lamp[15, 3]:=dword3.24;
Lamp[15, 4]:=dword4.24;
Lamp[15, 5]:=dword5.24;
Lamp[15, 6]:=dword6.24;
Lamp[15, 7]:=dword7.24;
Lamp[16, 0]:=dword0.23;
Lamp[16, 1]:=dword1.23;
Lamp[16, 2]:=dword2.23;
Lamp[16, 3]:=dword3.23;
Lamp[16, 4]:=dword4.23;
Lamp[16, 5]:=dword5.23;
Lamp[16, 6]:=dword6.23;
Lamp[16, 7]:=dword7.23;
Lamp[17, 0]:=dword0.22;
Lamp[17, 1]:=dword1.22;
Lamp[17, 2]:=dword2.22;
Lamp[17, 3]:=dword3.22;
Lamp[17, 4]:=dword4.22;
Lamp[17, 5]:=dword5.22;
Lamp[17, 6]:=dword6.22;
Lamp[17, 7]:=dword7.22;
Lamp[18, 0]:=dword0.21;
Lamp[18, 1]:=dword1.21;
Lamp[18, 2]:=dword2.21;
Lamp[18, 3]:=dword3.21;
Lamp[18, 4]:=dword4.21;
Lamp[18, 5]:=dword5.21;
Lamp[18, 6]:=dword6.21;
Lamp[18, 7]:=dword7.21;
Lamp[19, 0]:=dword0.20;
Lamp[19, 1]:=dword1.20;
Lamp[19, 2]:=dword2.20;
Lamp[19, 3]:=dword3.20;
Lamp[19, 4]:=dword4.20;
Lamp[19, 5]:=dword5.20;
Lamp[19, 6]:=dword6.20;
Lamp[19, 7]:=dword7.20;
Lamp[20, 0]:=dword0.19;
Lamp[20, 1]:=dword1.19;
Lamp[20, 2]:=dword2.19;
Lamp[20, 3]:=dword3.19;
Lamp[20, 4]:=dword4.19;
Lamp[20, 5]:=dword5.19;
Lamp[20, 6]:=dword6.19;
Lamp[20, 7]:=dword7.19;
Lamp[21, 0]:=dword0.18;
Lamp[21, 1]:=dword1.18;
Lamp[21, 2]:=dword2.18;
Lamp[21, 3]:=dword3.18;
Lamp[21, 4]:=dword4.18;
Lamp[21, 5]:=dword5.18;
Lamp[21, 6]:=dword6.18;
Lamp[21, 7]:=dword7.18;
Lamp[22, 0]:=dword0.17;
Lamp[22, 1]:=dword1.17;
Lamp[22, 2]:=dword2.17;
Lamp[22, 3]:=dword3.17;
Lamp[22, 4]:=dword4.17;
Lamp[22, 5]:=dword5.17;
Lamp[22, 6]:=dword6.17;
Lamp[22, 7]:=dword7.17;
Lamp[23, 0]:=dword0.16;
Lamp[23, 1]:=dword1.16;
Lamp[23, 2]:=dword2.16;
Lamp[23, 3]:=dword3.16;
Lamp[23, 4]:=dword4.16;
Lamp[23, 5]:=dword5.16;
Lamp[23, 6]:=dword6.16;
Lamp[23, 7]:=dword7.16;
Lamp[24, 0]:=dword0.16;
Lamp[24, 1]:=dword1.15;
Lamp[24, 2]:=dword2.15;
Lamp[24, 3]:=dword3.15;
Lamp[24, 4]:=dword4.15;
Lamp[24, 5]:=dword5.15;
Lamp[24, 6]:=dword6.15;
Lamp[24, 7]:=dword7.15;
Lamp[25, 0]:=dword0.14;
Lamp[25, 1]:=dword1.14;
Lamp[25, 2]:=dword2.14;
Lamp[25, 3]:=dword3.14;
Lamp[25, 4]:=dword4.14;
Lamp[25, 5]:=dword5.14;
Lamp[25, 6]:=dword6.14;
Lamp[25, 7]:=dword7.14;
Lamp[26, 0]:=dword0.13;
Lamp[26, 1]:=dword1.13;
Lamp[26, 2]:=dword2.13;
Lamp[26, 3]:=dword3.13;
Lamp[26, 4]:=dword4.13;
Lamp[26, 5]:=dword5.13;
Lamp[26, 6]:=dword6.13;
Lamp[26, 7]:=dword7.13;
Lamp[27, 0]:=dword0.12;
Lamp[27, 1]:=dword1.12;
Lamp[27, 2]:=dword2.12;
Lamp[27, 3]:=dword3.12;
Lamp[27, 4]:=dword4.12;
Lamp[27, 5]:=dword5.12;
Lamp[27, 6]:=dword6.12;
Lamp[27, 7]:=dword7.12;
Lamp[28, 0]:=dword0.11;
Lamp[28, 1]:=dword1.11;
Lamp[28, 2]:=dword2.11;
Lamp[28, 3]:=dword3.11;
Lamp[28, 4]:=dword4.11;
Lamp[28, 5]:=dword5.11;
Lamp[28, 6]:=dword6.11;
Lamp[28, 7]:=dword7.11;
Lamp[29, 0]:=dword0.10;
Lamp[29, 1]:=dword1.10;
Lamp[29, 2]:=dword2.10;
Lamp[29, 3]:=dword3.10;
Lamp[29, 4]:=dword4.10;
Lamp[29, 5]:=dword5.10;
Lamp[29, 6]:=dword6.10;
Lamp[29, 7]:=dword7.10;
Lamp[30, 0]:=dword0.9;
Lamp[30, 1]:=dword1.9;
Lamp[30, 2]:=dword2.9;
Lamp[30, 3]:=dword3.9;
Lamp[30, 4]:=dword4.9;
Lamp[30, 5]:=dword5.9;
Lamp[30, 6]:=dword6.9;
Lamp[30, 7]:=dword7.9;
Lamp[31, 0]:=dword0.8;
Lamp[31, 1]:=dword1.8;
Lamp[31, 2]:=dword2.8;
Lamp[31, 3]:=dword3.8;
Lamp[31, 4]:=dword4.8;
Lamp[31, 5]:=dword5.8;
Lamp[31, 6]:=dword6.8;
Lamp[31, 7]:=dword7.8;
Lamp[32, 0]:=dword0.7;
Lamp[32, 1]:=dword1.7;
Lamp[32, 2]:=dword2.7;
Lamp[32, 3]:=dword3.7;
Lamp[32, 4]:=dword4.7;
Lamp[32, 5]:=dword5.7;
Lamp[32, 6]:=dword6.7;
Lamp[32, 7]:=dword7.7;
Lamp[33, 0]:=dword0.6;
Lamp[33, 1]:=dword1.6;
Lamp[33, 2]:=dword2.6;
Lamp[33, 3]:=dword3.6;
Lamp[33, 4]:=dword4.6;
Lamp[33, 5]:=dword5.6;
Lamp[33, 6]:=dword6.6;
Lamp[33, 7]:=dword7.6;
Lamp[34, 0]:=dword0.5;
Lamp[34, 1]:=dword1.5;
Lamp[34, 2]:=dword2.5;
Lamp[34, 3]:=dword3.5;
Lamp[34, 4]:=dword4.5;
Lamp[34, 5]:=dword5.5;
Lamp[34, 6]:=dword6.5;
Lamp[34, 7]:=dword7.5;
Lamp[35, 0]:=dword0.4;
Lamp[35, 1]:=dword1.4;
Lamp[35, 2]:=dword2.4;
Lamp[35, 3]:=dword3.4;
Lamp[35, 4]:=dword4.4;
Lamp[35, 5]:=dword5.4;
Lamp[35, 6]:=dword6.4;
Lamp[35, 7]:=dword7.4;
Lamp[36, 0]:=dword0.3;
Lamp[36, 1]:=dword1.3;
Lamp[36, 2]:=dword2.3;
Lamp[36, 3]:=dword3.3;
Lamp[36, 4]:=dword4.3;
Lamp[36, 5]:=dword5.3;
Lamp[36, 6]:=dword6.3;
Lamp[36, 7]:=dword7.3;
Lamp[37, 0]:=dword0.2;
Lamp[37, 1]:=dword1.2;
Lamp[37, 2]:=dword2.2;
Lamp[37, 3]:=dword3.2;
Lamp[37, 4]:=dword4.2;
Lamp[37, 5]:=dword5.2;
Lamp[37, 6]:=dword6.2;
Lamp[37, 7]:=dword7.2;
Lamp[38, 0]:=dword0.1;
Lamp[38, 1]:=dword1.1;
Lamp[38, 2]:=dword2.1;
Lamp[38, 3]:=dword3.1;
Lamp[38, 4]:=dword4.1;
Lamp[38, 5]:=dword5.1;
Lamp[38, 6]:=dword6.1;
Lamp[38, 7]:=dword7.1;
Lamp[39, 0]:=dword0.0;
Lamp[39, 1]:=dword1.0;
Lamp[39, 2]:=dword2.0;
Lamp[39, 3]:=dword3.0;
Lamp[39, 4]:=dword4.0;
Lamp[39, 5]:=dword5.0;
Lamp[39, 6]:=dword6.0;
Lamp[39, 7]:=dword7.0;


          
END_PROGRAM

FUNCTION_BLOCK Tank_Model
  VAR_INPUT
    cfgTaskCycle : REAL;  (* Task cycle of the POU this model is running in miliseconds *)
    cfgLenght : REAL := 0;  (* Lenght of the tank in meters *)
    cfgWidth : REAL := 0;  (* Width of the tank in meters *)
    cfgHeight : REAL := 0;  (* Height of the tank in meters *)
    cfgStartLevel : REAL := 0;  (* Starting level of the tank in m~3 *)
    cfgFSHH : REAL := 95;  (* Float switch high high level in percentages of the volume of the tank *)
    cfgFSH : REAL := 80;  (* Float switch high level in percentages of the volume of the tank *)
    cfgFSL : REAL := 20;  (* Float switch low level in percentages of the volume of the tank *)
    cfgFSLL : REAL := 5;  (* Float switch low low level in percentages of the volume of the tank *)
    Inflow1 : REAL := 0;  (* Inflow, slot 1 to the tank in cubic meters per hour *)
    Inflow2 : REAL := 0;  (* Inflow, slot 2 to the tank in cubic meters per hour *)
    Inflow3 : REAL := 0;  (* Inflow, slot 3 to the tank in cubic meters per hour *)
    Inflow4 : REAL := 0;  (* Inflow, slot 4 to the tank in cubic meters per hour *)
    Inflow5 : REAL := 0;  (* Inflow, slot 5 to the tank in cubic meters per hour *)
    Outflow1 : REAL := 0;  (* Outflow, slot 1 to the tank in cubic meters per hour *)
    Outflow2 : REAL := 0;  (* Outflow, slot 2 to the tank in cubic meters per hour *)
    Outflow3 : REAL := 0;  (* Outflow, slot 3 to the tank in cubic meters per hour *)
    Outflow4 : REAL := 0;  (* Outflow, slot 4 to the tank in cubic meters per hour *)
    Outflow5 : REAL := 0;  (* Outflow, slot 5 to the tank in cubic meters per hour *)
  END_VAR
  VAR_OUTPUT
    TankLevel_cbm : REAL;  (* Tank level in cubic meters *)
    TankLevel_pc : REAL;  (* Tank level in percentages *)
    FSHHActive : BOOL;  (* Floating switch High high level active *)
    FSHActive : BOOL;  (* Floating switch High level active *)
    FSLActive : BOOL;  (* Floating switch Low level active *)
    FSLLActive : BOOL;  (* Floating switch Low low level active *)
  END_VAR
  VAR
    vNominalVolume : REAL;
    vInflowTotal : REAL;
    vOutflowTotal : REAL;
    vDeltaTime : REAL;
  END_VAR
  VAR RETAIN
    vColdRestart : BOOL;
  END_VAR

            IF NOT vColdRestart THEN
	TankLevel_cbm := cfgStartLevel;
	vColdRestart := TRUE;
END_IF

vNominalVolume := cfgLenght * cfgWidth * cfgHeight;

vInflowTotal := Inflow1 + Inflow2 + Inflow3 + Inflow4 + Inflow5;

vOutflowTotal := Outflow1 + Outflow2 + Outflow3 + Outflow4 + Outflow5;

(* Task cycle speed increase will lower the speed of TankLevel filling *)
vDeltaTime := cfgTaskCycle/DINT_TO_REAL(3600 * 1000);

(* Tank level calculation, independent of task execution cycle *)
TankLevel_cbm :=LIMIT(0,TankLevel_cbm + (vInflowTotal - vOutflowTotal) * vDeltaTime, vNominalVolume);

TankLevel_pc := (TankLevel_cbm / vNominalVolume) * 100;

(* Limit switch handling *)
FSHHActive := TankLevel_pc >= cfgFSHH;
FSHActive := TankLevel_pc >= cfgFSH;
FSLActive := TankLevel_pc <= cfgFSL;
FSLLActive := TankLevel_pc <= cfgFSLL;
          
END_FUNCTION_BLOCK

FUNCTION_BLOCK TankControl
  VAR_INPUT
    TankLevel_pc : REAL;
    LevelRef : REAL;
  END_VAR
  VAR_OUTPUT
    Drain : BOOL;
    Fill : BOOL;
  END_VAR

            IF LevelRef > TankLevel_pc + 2 THEN
	Fill := TRUE;
	Drain := FALSE;
ELSIF LevelRef < TankLevel_pc THEN
	Fill := FALSE;
	Drain := TRUE;
ELSE
	Fill:= FALSE;
	Drain:= FALSE;
END_IF
          
END_FUNCTION_BLOCK

PROGRAM MixingTank
  VAR
    vSystemState : DINT;
    vSequenceStarted : BOOL;
    vDrainingSequence : BOOL;
    SR : SR;
    NewSeqTimer : TON;
  END_VAR

            (* Logic part *)
(* Control the start and stop of the sequence *)
SR(Set1 := MixingTankGVL.PushButtonStart, Reset := MixingTankGVL.PushButtonStop, Q1 => vSequenceStarted);

(* If the tank is empty reset the DrainingSequence indication*)
IF MixingTankGVL.TankLevel <=0 THEN
	NewSeqTimer(IN:=TRUE, PT:=T#5S);
	IF NewSeqTimer.Q THEN
		vDrainingSequence := FALSE;
		NewSeqTimer(IN:=FALSE);
	END_IF
END_IF

//Use Tank level value to remember case machine state
IF vSequenceStarted THEN
	IF MixingTankGVL.TankLevel >= 0 AND MixingTankGVL.TankLevel <= 33 AND NOT vDrainingSequence THEN
		vSystemState := 0;
	END_IF
	
	IF MixingTankGVL.TankLevel >= 33 AND MixingTankGVL.TankLevel <= 66 AND NOT vDrainingSequence THEN
		vSystemState := 1;
	END_IF
	
	IF MixingTankGVL.TankLevel >= 66 AND MixingTankGVL.TankLevel < 95 AND NOT vDrainingSequence THEN
		vSystemState := 2;
	END_IF
	
	IF MixingTankGVL.TankLevel > 95 OR vDrainingSequence THEN
		vSystemState := 3;
	END_IF
ELSE
	vSystemState := 99;
END_IF


//Define the states logic
CASE vSystemState OF
	//First state. System below 33%
	0:
	MixingTankGVL.Pump1StartCmd := NOT MixingTankGVL.Pump1Running; //Start command pump 1 active until it starts
	MixingTankGVL.DrainValveCloseCmd := NOT MixingTankGVL.DrainValveClosed; //Close drain valve command active until it closes
	
	//Second state. System above 33%
	1:
	MixingTankGVL.Pump1StopCmd := MixingTankGVL.Pump1Running; //Stop command pump 1 active until it stops
	MixingTankGVL.Pump2StartCmd := NOT MixingTankGVL.Pump2Running; //Start command pump 2 active until it starts
	MixingTankGVL.DrainValveCloseCmd := NOT MixingTankGVL.DrainValveClosed; //Close drain valve command active until it closes
	
	//Third state. System above 66%
	2:
	MixingTankGVL.Pump2StopCmd := MixingTankGVL.Pump2Running; //Stop command pump 2 active until it stops
	MixingTankGVL.Pump1StartCmd := NOT MixingTankGVL.Pump1Running; //Start command pump 1 active until it starts
	MixingTankGVL.DrainValveCloseCmd := NOT MixingTankGVL.DrainValveClosed; //Close drain valve command active until it closes
	
	//Fourth state. System ready for draining
	3:
	vDrainingSequence := TRUE; //Draining sequence flag we set to true
	MixingTankGVL.Pump1StopCmd := MixingTankGVL.Pump1Running; //Stop command pump 1 active until it stops
	MixingTankGVL.Pump2StopCmd := MixingTankGVL.Pump2Running; //Stop command pump 2 active until it stops
	MixingTankGVL.DrainValveOpenCmd := NOT MixingTankGVL.DrainValveOpened; //Open drain valve command active until it opens
	
	//Sequence stopped state
	99:
	MixingTankGVL.Pump1StopCmd := MixingTankGVL.Pump1Running;
	MixingTankGVL.Pump2StopCmd := MixingTankGVL.Pump2Running;
	MixingTankGVL.DrainValveCloseCmd := NOT MixingTankGVL.DrainValveClosed;
END_CASE

          
END_PROGRAM

FUNCTION_BLOCK MoveSprite
  VAR_IN_OUT
    xCor : INT := 0;
    yCor : INT := 0;
  END_VAR
  VAR_INPUT
    xScreen : INT := 0;  (* Width of the screen *)
    yScreen : INT := 0;  (* Height of the screen *)
    SpriteWidth : INT := 0;  (* Width of the sprite *)
    SpriteHeight : INT := 0;  (* Height of the sprite *)
    ySpeed : INT := 0;  (* Control up or down movement with +- *)
    xSpeed : INT := 0;  (* Control left or right movement with +- *)
  END_VAR

            (* Reseting the position if sprite goes off screen *)
(* If moving left to right *)
IF xCor >= xScreen  AND xSpeed > 0 THEN
	xCor := -SpriteWidth;
(* If moving right to left *)
ELSIF xCor <= -SpriteWidth AND xSpeed < 0 THEN
	xCor := xScreen;	
END_IF
(* If moving from up, down *)
IF yCor >= yScreen AND ySpeed > 0 THEN
	yCor := -SpriteHeight;
(* If moving from down, up *)
ELSIF yCor < -SpriteHeight AND ySpeed < 0 THEN
	yCor := yScreen;	
END_IF

(* Actual moving of the coordinates *)
xCor := xCor + xSpeed;
yCor := yCor + ySpeed;

          
END_FUNCTION_BLOCK

FUNCTION_BLOCK Servo
  VAR_INPUT
    CmdFwd : BOOL := FALSE;
    CmdRev : BOOL := FALSE;
    PulseWidth : TIME := TIME#100ms;  (* Width of a pulse from the hall effect sensor when its above magnetic surface *)
  END_VAR
  VAR_OUTPUT
    S1 : BOOL := FALSE;
    S2 : BOOL := FALSE;
  END_VAR
  VAR
    tofS2 : TOF;
    tonS2 : TON;
    blink : BLINK;
    blinkOld : BOOL;
    vStartBlinker : BOOL;
  END_VAR

            vStartBlinker := (CmdFwd OR CmdRev) AND NOT (CmdFwd AND CmdRev);
Blink(ENABLE := vStartBlinker, TIMELOW:= PulseWidth, TIMEHIGH := PulseWidth);

tonS2(IN := blink.OUT, PT:=PulseWidth/2);
tofS2(IN := NOT tonS2.Q AND blinkOld, PT:=PulseWidth/2);
 
blinkOld := tonS2.Q;

IF CmdFwd THEN
	S1 := blink.OUT;
	S2 := tonS2.Q OR tofS2.Q;
ELSIF CmdRev THEN
	S1 := tonS2.Q OR tofS2.Q;
	S2 := blink.OUT;
END_IF
          
END_FUNCTION_BLOCK

PROGRAM Task02
  VAR
    PositionDetector : CTUD;
    PositionDetector2 : CTUD;
    vHorizontalCountS1 : DINT;
    vHorizontalCountS2 : DINT;
    vVerticalCountS1 : DINT;
    vVerticalCountS2 : DINT;
    rtHorizontalS1 : R_TRIG;
    rtHorizontalS2 : R_TRIG;
  END_VAR

            (* Quadrature signal array *)
rtHorizontalS1(CLK:=Task02GVl.HorizontalS1);
rtHorizontalS2(CLK:=Task02GVl.HorizontalS2);


PositionDetector2(
	CU:= rtHorizontalS2.Q, 
	CD:= FALSE, 
	CV=> vHorizontalCountS2);

PositionDetector(
	CU:= rtHorizontalS1.Q, 
	CD:= FALSE, 
	CV=> vHorizontalCountS1);
	
Task02GVL.HorizontalLeft := Task02GVL.ManLeft OR Task02GVl.ManUpLeft OR Task02GVl.ManDownLeft;
Task02GVL.HorizontalRight := Task02GVL.ManRight OR Task02GVl.ManUpRight OR Task02GVl.ManDownRight;
Task02GVL.VerticalUp := Task02GVL.ManUp OR Task02GVl.ManUpLeft OR Task02GVl.ManUpRight;
Task02GVL.VerticalDown := Task02GVL.ManDown OR Task02GVl.ManDownLeft OR Task02GVl.ManDownRight;
          
END_PROGRAM

PROGRAM Task03
  VAR
    vSequenceA : DINT := 1;
    TimerA : TOF;
    vSequenceB : DINT := 0;
    TimerB : TOF;
    Start : BOOL;
    StartOld : BOOL;
    vSequence : DINT := 0;
    TactTimer : TON;
    vPeriodTime : TIME := TIME#1m25s0ms;
    vElapsedTime : TIME;
  END_VAR

            
TactTimer(IN:=TRUE, PT:=vPeriodTime, ET => vElapsedTime);
IF TactTimer.Q THEN
	TactTimer(IN:=FALSE);
END_IF
(* Direction Up, Down traffic light *)
Task03GVL.TLight3Red := vElapsedTime <= T#5S OR vElapsedTime >= T#37S AND vElapsedTime <= T#85S;
Task03GVL.TLight3Yellow := vElapsedTime > T#3S AND vElapsedTime <= T#5S OR vElapsedTime >= T#35S AND vElapsedTime <= T#37S;
Task03GVL.TLight3Green := vElapsedTime >= T#5S AND vElapsedTime <= T#35S;

(* Mirror the other side of the Up, Down direction *)
Task03GVL.TLight4Red := Task03GVL.TLight3Red;
Task03GVL.TLight4Yellow := Task03GVL.TLight3Yellow;
Task03GVL.TLight4Green := Task03GVL.TLight3Green;

(* Direction Left, Right traffic light *)
Task03GVL.TLight2Red := vElapsedTime >= T#0S AND vElapsedTime <= T#39S OR vElapsedTime >= T#71S AND vElapsedTime <= T#85S;
Task03GVL.TLight2Yellow := vElapsedTime > T#37S AND vElapsedTime <= T#39S OR vElapsedTime >= T#69S AND vElapsedTime <= T#71S;
Task03GVL.TLight2Green := vElapsedTime >= T#39S AND vElapsedTime <= T#69S;

(* Mirror the other side of the Left, Right direction *)
Task03GVL.TLight1Red := Task03GVL.TLight2Red;
Task03GVL.TLight1Yellow := Task03GVL.TLight2Yellow;
Task03GVL.TLight1Green := Task03GVL.TLight2Green;
(*CASE vSequence OF
	0:
	(* Starting sequence, direction Up, Down *)
	TimerA
	Task03GVL.TLight1Red := TRUE;
	
END_CASE
CASE vSequenceA OF
	0: TimerA(IN:=FALSE,PT:=T#20S);
	Task03GVL.TLight1Yellow:= FALSE;
	Task03GVL.TLight1Red:= FALSE;
	Task03GVL.TLight1Green:= TimerA.Q;
	Task03GVL.TLight2Green := Task03GVL.TLight1Green;
	IF NOT TimerA.Q THEN
		TimerA(IN:=TRUE);
		vSequenceA:=1;
	END_IF
	1: TimerA(IN:=FALSE,PT:=T#4S);
	Task03GVL.TLight1Red:= FALSE;
	Task03GVL.TLight1Green:= FALSE;
	Task03GVL.TLight1Yellow:= TimerA.Q;
	Task03GVL.TLight2Yellow := Task03GVL.TLight1Yellow;
	IF NOT TimerA.Q THEN
		TimerA(IN:=TRUE);
		vSequenceA:=2;
	END_IF
		2: TimerA(IN:=FALSE,PT:=T#30S);
	Task03GVL.TLight1Green:= FALSE;
	Task03GVL.TLight1Yellow:= FALSE;
	Task03GVL.TLight1Red:= TimerA.Q;
	Task03GVL.TLight2Red := Task03GVL.TLight1Red;
	IF NOT TimerA.Q THEN
		TimerA(IN:=TRUE);
		vSequenceA:=3;
	END_IF
		3: TimerA(IN:=FALSE,PT:=T#4S);
	Task03GVL.TLight1Green:= FALSE;
	Task03GVL.TLight1Red:= TimerA.Q;
	Task03GVL.TLight1Yellow:= TimerA.Q;
	Task03GVL.TLight2Red := Task03GVL.TLight1Red;
	Task03GVL.TLight2Yellow := Task03GVL.TLight1Yellow;
	IF NOT TimerA.Q THEN
		TimerA(IN:=TRUE);
		vSequenceA:=0;
		IF vSequenceB=6 THEN
		vSequenceB:=3;	
		END_IF
		
	END_IF
END_CASE

CASE vSequenceB OF
	0: TimerB(IN:=FALSE,PT:=T#4S);
	Task03GVL.TLight3Green:= FALSE;
	Task03GVL.TLight3Red:= TimerB.Q;
	Task03GVL.TLight3Yellow:= TimerB.Q;
	Task03GVL.TLight4Red := Task03GVL.TLight3Red;
	Task03GVL.TLight4Yellow := Task03GVL.TLight3Yellow;
	IF NOT TimerB.Q THEN
		TimerB(IN:=TRUE);
		vSequenceB:=1;
	END_IF
	
	1: TimerB(IN:=FALSE,PT:=T#20S);
	Task03GVL.TLight3Yellow:= FALSE;
	Task03GVL.TLight3Red:= FALSE;
	Task03GVL.TLight3Green:= TimerB.Q;
	Task03GVL.TLight4Green := Task03GVL.TLight3Green;
	IF NOT TimerB.Q THEN
		TimerB(IN:=TRUE);
		vSequenceB:=2;
	END_IF
	
	2: TimerB(IN:=FALSE,PT:=T#4S);
	Task03GVL.TLight3Red:= FALSE;
	Task03GVL.TLight3Green:= FALSE;
	Task03GVL.TLight3Yellow:= TimerB.Q;
	Task03GVL.TLight4Yellow := Task03GVL.TLight3Yellow;
	IF NOT TimerB.Q THEN
		TimerB(IN:=TRUE);
		vSequenceB:=3;
	END_IF
	
		3: TimerB(IN:=FALSE,PT:=T#30S);
	Task03GVL.TLight3Green:= FALSE;
	Task03GVL.TLight3Yellow:= FALSE;
	Task03GVL.TLight3Red:= TimerB.Q;
	Task03GVL.TLight4Red := Task03GVL.TLight3Red;
	IF NOT TimerB.Q THEN
		TimerB(IN:=TRUE);
		vSequenceB:=0;
	END_IF
		
END_CASE
END_IF;*)
          
END_PROGRAM

PROGRAM Task04
  VAR
    M3 : BOOL;
    Start_Desno : BOOL;
    Start_Lijevo : BOOL;
    STOP : BOOL;
    SklopkaPreopterecenja : BOOL;
    M3_Lijevo : BOOL;
    M3_Desno : BOOL;
    Cooling : TOF;
    StreliceLijevoInv : BOOL;
    StreliceDesnoInv : BOOL;
  END_VAR

            (*Zadatak 4.
Promena smera obrtanja trofaznog asinhronog motora izvodi se promenom redosleda faza napona
napajanja motora. Upravljanje motorom izvodi se tasterima "START-DESNO", "START-LEVO" i "STOP".
Motor se sem toga štiti i od preopterećenja motornom zaštitnom sklopkom.
Razraditi rešenje kašnjenja sa PLC kontrolerom.*)

M3_Lijevo:=(M3_Lijevo OR Start_Lijevo) AND NOT M3_Desno AND NOT STOP AND NOT SklopkaPreopterecenja AND NOT Cooling.Q;
M3_Desno:=(M3_Desno OR Start_Desno) AND NOT M3_Lijevo AND NOT STOP AND NOT SklopkaPreopterecenja AND NOT Cooling.Q;

M3:= M3_Lijevo OR M3_Desno; (*Ovo je samo simulirani motor jer nemamo pravi*)
Cooling(IN:=Stop, PT:=T#5S);
StreliceLijevoInv:=M3_Desno OR (NOT M3_Desno AND NOT M3_Lijevo);
StreliceDesnoInv:=M3_Lijevo OR (NOT M3_Desno AND NOT M3_Lijevo);
          
END_PROGRAM

PROGRAM Task05

            
          
END_PROGRAM

PROGRAM Task06

            IF Task06GVL.EmcyStop THEN
	Task06GVL.CraneDown := Task06GVL.JoyDown OR Task06GVL.JoyDownLeft OR Task06GVL.JoyDownRight;
	Task06GVL.CraneUp := Task06GVL.JoyUp OR Task06GVL.JoyUpLeft OR Task06GVL.JoyUpRight;

	Task06GVL.MotorRight := Task06GVL.JoyRight OR Task06GVL.JoyUpRight OR Task06GVL.JoyDownRight;
	Task06GVL.MotorLeft := Task06GVL.JoyLeft OR Task06GVL.JoyUpLeft OR Task06GVL.JoyDownLeft;
ELSE
	Task06GVL.CraneDown := FALSE;
	Task06GVL.CraneUp := FALSE;

	Task06GVL.MotorRight := FALSE;
	Task06GVL.MotorLeft := FALSE;
END_IF




          
END_PROGRAM

PROGRAM Task07
  VAR
    StartRight : BOOL := FALSE;
    StartLeft : BOOL := FALSE;
    PulseWidth : TIME := TIME#100ms;  (* Width of a pulse from the hall effect sensor when its above magnetic surface *)
    tofS2 : TOF;
    tonS2 : TON;
    blinkS1 : BLINK;
    blinkS1Old : BOOL;
    S1 : BOOL := FALSE;
    S2 : BOOL := FALSE;
  END_VAR

            blinkS1(ENABLE := StartRight OR StartLeft, TIMELOW:= PulseWidth, TIMEHIGH := PulseWidth);
tonS2(IN := blinkS1.OUT, PT:=PulseWidth/2);
tofS2(IN := NOT tonS2.Q AND blinkS1Old, PT:=PulseWidth/2);
 
blinkS1Old := tonS2.Q;

S1 := blinkS1.OUT;
S2 := tonS2.Q OR tofS2.Q;
          
END_PROGRAM

PROGRAM Task08

            
          
END_PROGRAM

PROGRAM Task09

            
          
END_PROGRAM

PROGRAM Task10

            
          
END_PROGRAM

PROGRAM Task01Sim
  VAR
    Pump1Sim : Pump_Model;  (* Simulator and graphics *)
    Pump2Sim : Pump_Model;
    DrainValveSim : OnOffValve_model;
    MixingTank : Tank_Model;
    vPump1RunningDint : DINT;
    vPump2RunningDint : DINT;
    vPump1FlowRate : REAL;
    vPump2FlowRate : REAL;
    ValveIcon : STRING;
    Pump1Icon : STRING;
    Pump2Icon : STRING;
  END_VAR

            (*Task 01 Simulator*)
Pump1Sim(
	OnCmd:= MixingTankGVL.Pump1StartCmd, 
	OffCmd:= MixingTankGVL.Pump1StopCmd, 
	cfgFlowrate:= 1200, 
	RunStatus=> vPump1RunningDint, 
	FlowmeterOut=> vPump1FlowRate);
MixingTankGVL.Pump1Running:= DINT_TO_BOOL(vPump1RunningDint);
	
Pump2Sim(
	OnCmd:= MixingTankGVL.Pump2StartCmd, 
	OffCmd:= MixingTankGVL.Pump2StopCmd, 
	cfgFlowrate:= 1200, 
	RunStatus=> vPump2RunningDint, 
	FlowmeterOut=> vPump2FlowRate);
MixingTankGVL.Pump2Running:= DINT_TO_BOOL(vPump2RunningDint);
	
DrainValveSim(
	OpenCmd:= MixingTankGVL.DrainValveOpenCmd, 
	CloseCmd:= MixingTankGVL.DrainValveCloseCmd, 
	cfgOpeningTime:= T#2S, 
	cfgClosingTime:= T#2S, 
	Opened=> MixingTankGVL.DrainValveOpened, 
	Closed=> MixingTankGVL.DrainValveClosed);

MixingTank(
	cfgTaskCycle:= 100, 
	cfgLenght:= 5, 
	cfgWidth:= 5, 
	cfgHeight:= 5, 
	cfgStartLevel:= 0, 
	Inflow1:= vPump1FlowRate, 
	Inflow2:= vPump2FlowRate, 
	Outflow1:= 2400*BOOL_TO_REAL(MixingTankGVL.DrainValveOpened), 
	TankLevel_pc=> MixingTankGVL.TankLevel);
	
IF MixingTankGVL.DrainValveClosed THEN
	ValveIcon := 'Valve1';
ELSIF MixingTankGVL.DrainValveOpened THEN
	ValveIcon := 'Valve2';
ELSE
	ValveIcon := 'Valve3';
END_IF

IF MixingTankGVL.Pump1Running THEN
	Pump1Icon := 'PumpOn';
ELSE
	Pump1Icon := 'PumpOff';
END_IF

IF MixingTankGVL.Pump2Running THEN
	Pump2Icon := 'PumpOn';
ELSE
	Pump2Icon := 'PumpOff';
END_IF


          
END_PROGRAM

PROGRAM Task02Sim
  VAR
    HorizontalAxis : Servo;
    VerticalAxis : Servo;
    rtHIncrement : R_TRIG;
    rtHDecrement : R_TRIG;
    rtVIncrement : R_TRIG;
    rtVDecrement : R_TRIG;
    vHorizontalS1Old : BOOL;
    vHorizontalS2Old : BOOL;
    vVerticalS1Old : BOOL;
    vVerticalS2Old : BOOL;
    PositionCounterVerticalAxis : CTUD;
    vHorizontalPos : DINT;
    PositionCounterHorizontalAxis : CTUD;
    vVerticalPos : WORD;
    vPositionX : REAL;
    vPositionY : REAL;
    vResetSIM : BOOL;
    vHorizontalLimit : BOOL;
    vVerticalLimit : BOOL;
  END_VAR

            (* The actual servos that move the watering equipment *)
vHorizontalLimit := vPositionX >= 940;
vVerticalLimit := vPositionY >= 500;

(* Maximum range - 940 steps *)
HorizontalAxis(
	CmdFwd:= Task02GVL.HorizontalRight AND NOT vHorizontalLimit, 
	CmdRev:= Task02GVL.HorizontalLeft, 
	PulseWidth:= T#0.1S , 
	S1=> Task02GVL.HorizontalS1, 
	S2=> Task02GVL.HorizontalS2);
	
(* Maximum range - 500 steps *)	
VerticalAxis(
	CmdFwd:= Task02GVL.VerticalDown AND NOT vVerticalLimit, 
	CmdRev:= Task02GVL.VerticalUp, 
	PulseWidth:= T#0.1S , 
	S1=> Task02GVL.VerticalS1, 
	S2=> Task02GVL.VerticalS2);

IF vResetSIM THEN
	vHorizontalPos := 0;
	vVerticalPos := 0;
END_IF

IF Task02GVL.HorizontalS1 <> vHorizontalS1Old THEN
	IF Task02GVL.HorizontalS1 <> Task02GVL.HorizontalS2 THEN
		rtHIncrement(CLK:=TRUE);
	ELSE
		rtHDecrement(CLK:=TRUE);
	END_IF
ELSE
	rtHIncrement(CLK:=FALSE);
	rtHDecrement(CLK:=FALSE);
END_IF

IF Task02GVL.VerticalS1 <> vVerticalS1Old THEN
	IF Task02GVL.VerticalS1 <> Task02GVL.VerticalS2 THEN
		rtVIncrement(CLK:=TRUE);
	ELSE
		rtVDecrement(CLK:=TRUE);
	END_IF
ELSE
	rtVIncrement(CLK:=FALSE);
	rtVDecrement(CLK:=FALSE);
END_IF

PositionCounterHorizontalAxis(
	CU:= rtHIncrement.Q, 
	CD:= rtHDecrement.Q, 
	CV=> vHorizontalPos);

PositionCounterVerticalAxis(
	CU:= rtVIncrement.Q, 
	CD:= rtVDecrement.Q, 
	CV=> vVerticalPos);
	
(* Position of the system *)
(* For every 5 pulses we move 200 px *)
vPositionX := (DINT_TO_REAL(vHorizontalPos)/ 5) * 200;
vPositionY := (DINT_TO_REAL(vVerticalPos)/ 5) * 200;
	
vHorizontalS1Old := Task02GVL.HorizontalS1;
vVerticalS1Old := Task02GVL.VerticalS1;
          
END_PROGRAM

PROGRAM Task03Sim
  VAR
    Car1X : INT := 925;  (* Red car *)
    Car1Y : INT := 740;
    Car1Width : INT := 100;
    Car1Height : INT := 230;
    Car2X : INT := 420;  (* Blue car *)
    Car2Y : INT := 511;
    Car2Width : INT := 230;
    Car2Height : INT := 100;
    Car3X : INT := 1160;  (* Green car *)
    Car3Y : INT := 366;
    Car3Width : INT := 230;
    Car3Height : INT := 100;
    Car4X : INT := 775;  (* Yellow car *)
    Car4Y : INT := 0;
    Car4Width : INT := 100;
    Car4Height : INT := 230;
    Speed : INT := 25;
    vCarCrash : BOOL;
    vReset : BOOL;
    xExplosion : INT;
    yExplosion : INT;
    Car3Car4Coll : CollisionDetection;
    Car3Car1Coll : CollisionDetection;
    Car2Car1Coll : CollisionDetection;
    Car2Car4Coll : CollisionDetection;
    MoveCar1 : MoveSprite;
    MoveCar2 : MoveSprite;
    MoveCar3 : MoveSprite;
    MoveCar4 : MoveSprite;
  END_VAR

            (* Collision detection *)
(* Car3 and Car 4 *)
Car3Car4Coll(
	xcor1:= Car3X, 
	ycor1:= Car3Y, 
	height1:= Car3Height, 
	width1:= Car3Width, 
	xcor2:= Car4X, 
	ycor2:= Car4Y, 
	height2:= Car4Height, 
	width2:= Car4Width);
(* Car3 and Car 1 *)
Car3Car1Coll(
	xcor1:= Car3X, 
	ycor1:= Car3Y, 
	height1:= Car3Height, 
	width1:= Car3Width, 
	xcor2:= Car1X, 
	ycor2:= Car1Y, 
	height2:= Car1Height, 
	width2:= Car1Width);
(* Car2 and Car 4 *)
Car2Car4Coll(
	xcor1:= Car2X, 
	ycor1:= Car2Y, 
	height1:= Car2Height, 
	width1:= Car2Width, 
	xcor2:= Car4X, 
	ycor2:= Car4Y, 
	height2:= Car4Height, 
	width2:= Car4Width);
(* Car2 and Car 1 *)
Car2Car1Coll(
	xcor1:= Car2X, 
	ycor1:= Car2Y, 
	height1:= Car2Height, 
	width1:= Car2Width, 
	xcor2:= Car1X, 
	ycor2:= Car1Y, 
	height2:= Car1Height, 
	width2:= Car1Width);

IF Car3Car4Coll.isCollision OR Car3Car1Coll.isCollision OR Car2Car4Coll.isCollision OR Car2Car1Coll.isCollision THEN
	vCarCrash := TRUE;
ELSE
	vCarCrash := FALSE;	
END_IF

(* Explosion graphic *)
IF Car3Car4Coll.isCollision THEN
	xExplosion := Car3X;
	yExplosion := Car3Y;
ELSIF Car3Car1Coll.isCollision THEN
	xExplosion := Car3X;
	yExplosion := Car3Y;
ELSIF Car2Car4Coll.isCollision THEN
	xExplosion := Car2X + Car2Width;
	yExplosion := Car2Y;
ELSIF Car2Car1Coll.isCollision THEN
	xExplosion := Car2X + Car2Width;
	yExplosion := Car2Y;
ELSE
	xExplosion := 2000;
	yExplosion := 2000;
END_IF

(* Car movements *)
IF  vCarCrash THEN
	//wait
	IF vReset THEN
		(* Reset to start position *)
		Car1X:= 925;
		Car1Y:= 740;
		Car2X:= 420;
		Car2Y:= 511;
		Car3X:= 1160;
		Car3Y:= 366;
		Car4X:= 775;
		Car4Y:= 0;
	END_IF
ELSE
	(* Define what cars do depending on lights *)
	(* car moves if its green for him or he is past the traffic ligght but stops at the traffic light if its red, or yellow.*)
	IF Task03GVL.TLight4Green OR Car1Y - 740 < 0 OR Car1Y - 740 > Speed THEN
		MoveCar1(
		xCor:= Car1X, 
		yCor:= Car1Y, 
		xScreen:= 1830, 
		yScreen:= 930,
		SpriteWidth:= Car1Width, 
		SpriteHeight:= Car1Height, 
		ySpeed:= -Speed, 
		xSpeed:= 0 );
	END_IF;
	IF Task03GVL.TLight2Green OR Car2X - 420 < 0 OR Car2X - 420 > Speed THEN
		MoveCar2(
		xCor:= Car2X, 
		yCor:= Car2Y, 
		xScreen:= 1830, 
		yScreen:= 930,
		SpriteWidth:= Car2Width, 
		SpriteHeight:= Car2Height,  
		ySpeed:= 0, 
		xSpeed:= Speed );
	END_IF;
	IF Task03GVL.TLight1Green OR Car3X - 1160 < 0 OR Car3X - 1160 > Speed THEN
		MoveCar3(
		xCor:= Car3X, 
		yCor:= Car3Y, 
		xScreen:= 1830, 
		yScreen:= 930,
		SpriteWidth:= Car3Width, 
		SpriteHeight:= Car3Height,  
		ySpeed:= 0, 
		xSpeed:= -Speed );
	END_IF;
	IF Task03GVL.TLight3Green OR Car4Y - 0 < 0 OR Car4Y - 0 > Speed THEN
		MoveCar4(
		xCor:= Car4X, 
		yCor:= Car4Y, 
		xScreen:= 1830, 
		yScreen:= 930,
		SpriteWidth:= Car4Width, 
		SpriteHeight:= Car4Height,  
		ySpeed:= Speed, 
		xSpeed:= 0 );
	END_IF;
END_IF


          
END_PROGRAM

PROGRAM Task04Sim

            
          
END_PROGRAM

PROGRAM Task05Sim
  VAR
    vConveyorElements : ARRAY[0..31] OF DINT;
    vBottleImage : ARRAY[0..31] OF STRING;
    vBox : ARRAY[0..23] OF DINT;
    vBoxBottleImage : ARRAY[0..23] OF STRING;
    i : INT;
    ArrayShifter : ShiftArray;
    TactGenerator : BLINK;
    vShift : BOOL;
    vRandomNumber : INT;
    vPlaceNewBottle : BOOL;
    vNewBottle : INT;
    ShiftTrig : R_TRIG;
    vBoxSum : REAL;
    vBoxFull : BOOL;
    vPackageEfficiency : REAL;
    vBoxValue : REAL;
    vBrokenBottleDetected : BOOL;
  END_VAR

            vRandomNumber := vRandomNumber + 1;
IF vRandomNumber > 4 THEN
	vRandomNumber := 0;
END_IF
TactGenerator(ENABLE:= TRUE, TIMELOW:= T#0.5S, TIMEHIGH:= T#0.5S, OUT=>vShift );
ShiftTrig(CLK:=vShift);

IF ShiftTrig.Q THEN
	vNewBottle := vRandomNumber;
ELSE
	vNewBottle := 0;
END_IF

